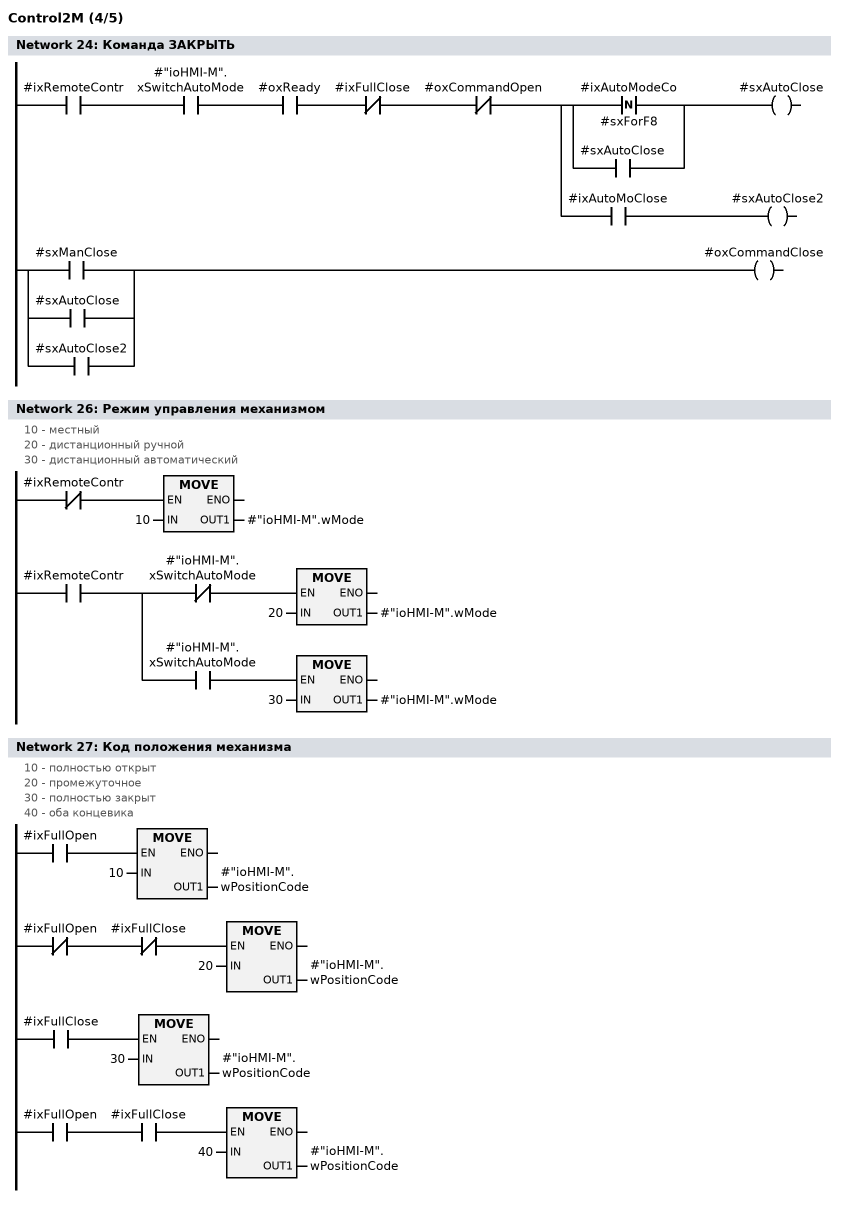
   RUNG wire#powerrail
      Contact( #ixRemoteContr )
      Contact( #"ioHMI-M".xSwitchAutoMode )
      Contact( #oxReady )
      I_Contact( #ixFullClose )
      I_Contact( #oxCommandOpen )
      wire#w1
      N_Contact(operand := #ixAutoModeCo, bit := #sxForF8)
      wire#w2
      Coil( #sxAutoClose )
   END_RUNG
   RUNG wire#w1
      Contact( #sxAutoClose )
   END_RUNG wire#w2
   RUNG wire#w1
      Contact( #ixAutoMoClose )
      Coil( #sxAutoClose2 )
   END_RUNG
   RUNG wire#powerrail
      Contact( #sxManClose )
      wire#w3
      Coil( #oxCommandClose )
   END_RUNG
   RUNG wire#powerrail
      Contact( #sxAutoClose )
   END_RUNG wire#w3
   RUNG wire#powerrail
      Contact( #sxAutoClose2 )
   END_RUNG wire#w3
   // the same network as SCL:
   #_w1 := #ixRemoteContr AND #"ioHMI-M".xSwitchAutoMode AND #oxReady AND NOT #ixFullClose AND NOT #oxCommandOpen;
   #_w2 := #_w1 AND NOT #ixAutoModeCo AND #sxForF8;   // falling edge of #ixAutoModeCo
   #sxForF8 := #ixAutoModeCo;
   #sxAutoClose := #_w2 OR (#_w1 AND #sxAutoClose);
   #sxAutoClose2 := #_w1 AND #ixAutoMoClose;
   #oxCommandClose := #sxManClose OR #sxAutoClose OR #sxAutoClose2;
END_REGION

REGION Network 26: Режим управления механизмом
   // 10 - местный
   // 20 - дистанционный ручной
   // 30 - дистанционный автоматический
   RUNG wire#powerrail
      I_Contact( #ixRemoteContr )
      Move(in := 10, out1 => #"ioHMI-M".wMode)
   END_RUNG
   RUNG wire#powerrail
      Contact( #ixRemoteContr )
      wire#w1
      I_Contact( #"ioHMI-M".xSwitchAutoMode )
      Move(in := 20, out1 => #"ioHMI-M".wMode)
   END_RUNG
   RUNG wire#w1
      Contact( #"ioHMI-M".xSwitchAutoMode )
      Move(in := 30, out1 => #"ioHMI-M".wMode)
   END_RUNG
   // the same network as SCL:
   IF NOT #ixRemoteContr THEN #"ioHMI-M".wMode := 10; END_IF;
   IF #ixRemoteContr AND NOT #"ioHMI-M".xSwitchAutoMode THEN #"ioHMI-M".wMode := 20; END_IF;
   IF #ixRemoteContr AND #"ioHMI-M".xSwitchAutoMode THEN #"ioHMI-M".wMode := 30; END_IF;
END_REGION

REGION Network 27: Код положения механизма
   // 10 - полностью открыт
   // 20 - промежуточное
   // 30 - полностью закрыт
   // 40 - оба концевика
   RUNG wire#powerrail
      Contact( #ixFullOpen )
      Move(in := 10, out1 => #"ioHMI-M".wPositionCode)
   END_RUNG
   RUNG wire#powerrail
      I_Contact( #ixFullOpen )
      I_Contact( #ixFullClose )
      Move(in := 20, out1 => #"ioHMI-M".wPositionCode)
   END_RUNG
   RUNG wire#powerrail
      Contact( #ixFullClose )
      Move(in := 30, out1 => #"ioHMI-M".wPositionCode)
   END_RUNG
   RUNG wire#powerrail
      Contact( #ixFullOpen )
      Contact( #ixFullClose )
      Move(in := 40, out1 => #"ioHMI-M".wPositionCode)
   END_RUNG
   // the same network as SCL:
   IF #ixFullOpen THEN #"ioHMI-M".wPositionCode := 10; END_IF;
   IF NOT #ixFullOpen AND NOT #ixFullClose THEN #"ioHMI-M".wPositionCode := 20; END_IF;
   IF #ixFullClose THEN #"ioHMI-M".wPositionCode := 30; END_IF;
   IF #ixFullOpen AND #ixFullClose THEN #"ioHMI-M".wPositionCode := 40; END_IF;
END_REGION

REGION Network 28: Код управления механизмом
   // 10 - нет команды на ход механизма
   // 20 - команда открыть
   // 30 - команда закрыть
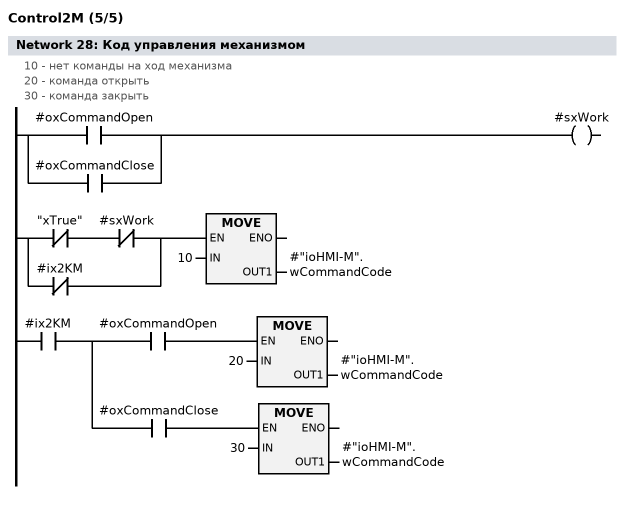
   RUNG wire#powerrail
      Contact( #oxCommandOpen )
      wire#w1
      Coil( #sxWork )
   END_RUNG
   RUNG wire#powerrail
      Contact( #oxCommandClose )
   END_RUNG wire#w1
   RUNG wire#powerrail
      I_Contact( "xTrue" )
      I_Contact( #sxWork )
      wire#w2
      Move(in := 10, out1 => #"ioHMI-M".wCommandCode)
   END_RUNG
   RUNG wire#powerrail
      I_Contact( #ix2KM )
   END_RUNG wire#w2
   RUNG wire#powerrail
      Contact( #ix2KM )
      wire#w3
      Contact( #oxCommandOpen )
      Move(in := 20, out1 => #"ioHMI-M".wCommandCode)
   END_RUNG
   RUNG wire#w3
      Contact( #oxCommandClose )
      Move(in := 30, out1 => #"ioHMI-M".wCommandCode)
   END_RUNG
   // the same network as SCL:
   #sxWork := #oxCommandOpen OR #oxCommandClose;
   IF (NOT "xTrue" AND NOT #sxWork) OR NOT #ix2KM THEN #"ioHMI-M".wCommandCode := 10; END_IF;
   IF #ix2KM AND #oxCommandOpen THEN #"ioHMI-M".wCommandCode := 20; END_IF;
   IF #ix2KM AND #oxCommandClose THEN #"ioHMI-M".wCommandCode := 30; END_IF;
END_REGION
END_FUNCTION_BLOCK

FUNCTION_BLOCK "ControlGate"   // FB503, LAD
{ S7_Optimized_Access := 'TRUE' }
VERSION : 0.1
   VAR_INPUT
      ixGateReady : Bool;   // Готовность шлюзового затвора
      ixRemoteContr : Bool;   // Ключ в положении Дистанц. рехим
      ixXKM : Bool;   // Пускатель включен
      ixExtStop : Bool;   // Внешняя блокировка
      ixAutoModeCommand : Bool;   // Авт.режим, 1=открыть, 0=закрыть
   END_VAR
   VAR_OUTPUT
      oxButSTART : Bool;   // Кнопка ПУСК ручного режима
      oxButSTOP : Bool;   // Кнопка СТОП ручного режима
      oxSwitchAutoMode : Bool;   // Переключатель (автомат.=1, ручной=0) на ЧМИ
      oxReady : Bool;   // Готовность механизма
      oxCommandOn : Bool;   // Команда Пуск
   END_VAR
   VAR_IN_OUT
      "ioHMI-M" : "uHMI-Machine";   // Структура данных связи с ЧМИ
   END_VAR
   VAR
      sxWarning : Bool;   // Есть предупреждения
      sxFault : Bool;   // Есть авария
      sxWork : Bool;   // Есть моя команда
      sxForF1 : Bool;   // Статический бит для обнаружения фронта сигнала
      sxForF6 : Bool;   // Статический бит для обнаружения фронта сигнала
      sxForF7 : Bool;   // Статический бит для обнаружения фронта сигнала
      IEC_TimerInstance2 : TON_TIME;   // Таймер
      IEC_TimerInstance1 : TON_TIME;   // Таймер
      sxManStart : Bool;   // Статический бит для команды ручного режима
      sxAutoStart : Bool;   // Статический бит для команды автоматического режима
   END_VAR
   VAR_TEMP
      tx1 : Bool;   // Временный бит
      tx2 : Bool;
   END_VAR
   VAR_TEMP   // added for the SCL form of the ladder/FBD networks
      _w1 : Bool;
      _w2 : Bool;
   END_VAR
BEGIN

REGION Network 4: Подготовка данных от HMI:
END_REGION

REGION Network 5 (SCL): -виртуальные кнопки
   #oxButSTART  :=  #"ioHMI-M".xButManOpen;
   #oxButSTOP :=  #"ioHMI-M".xButManClose;

   #oxSwitchAutoMode := #"ioHMI-M".xSwitchAutoMode;
END_REGION

REGION Network 7: ПРЕДУПРЕЖДЕНИЯ 3М-8М (для журнала предупреждений на ЧМИ)
   // //wWarnings.%X0 - полностью закрыт
   // //wWarnings.%X1 - полностью открыт
   // wWarnings.%X2 - нет готовности от механизма (было в дистанционном режиме, с 27.12.2020 - во всех режимах)
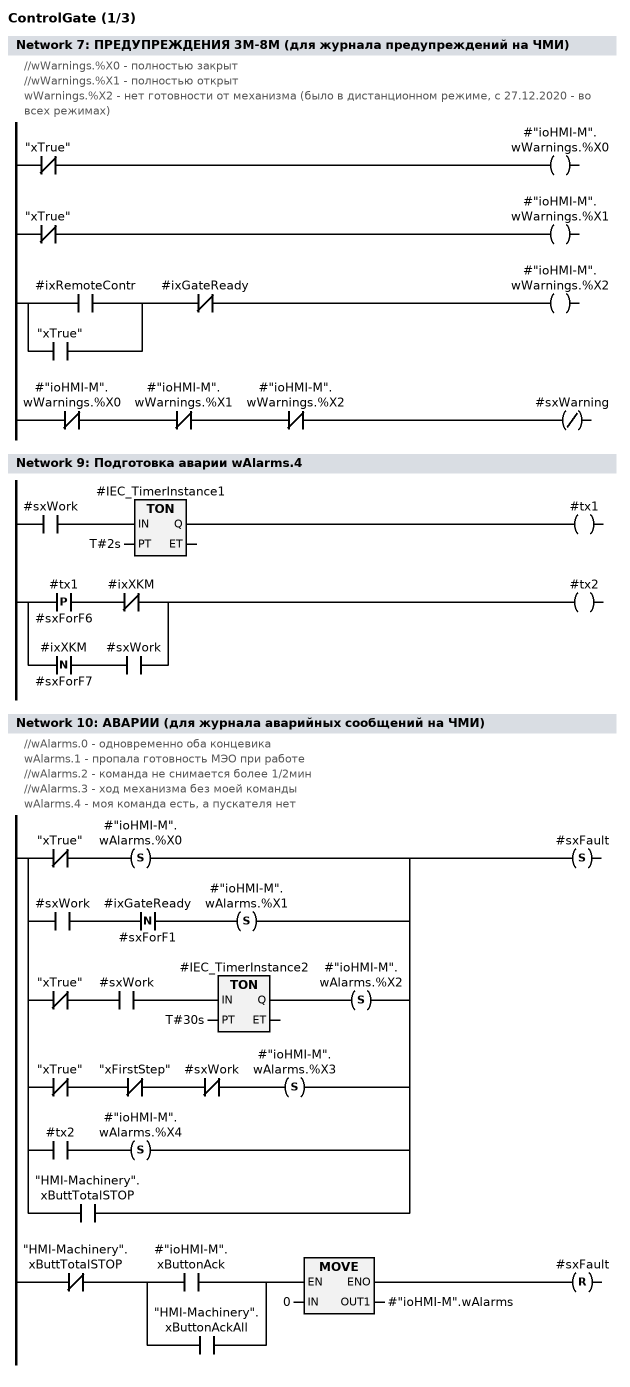
   RUNG wire#powerrail
      I_Contact( "xTrue" )
      Coil( #"ioHMI-M".wWarnings.%X0 )
   END_RUNG
   RUNG wire#powerrail
      I_Contact( "xTrue" )
      Coil( #"ioHMI-M".wWarnings.%X1 )
   END_RUNG
   RUNG wire#powerrail
      Contact( #ixRemoteContr )
      wire#w1
      I_Contact( #ixGateReady )
      Coil( #"ioHMI-M".wWarnings.%X2 )
   END_RUNG
   RUNG wire#powerrail
      Contact( "xTrue" )
   END_RUNG wire#w1
   RUNG wire#powerrail
      I_Contact( #"ioHMI-M".wWarnings.%X0 )
      I_Contact( #"ioHMI-M".wWarnings.%X1 )
      I_Contact( #"ioHMI-M".wWarnings.%X2 )
      I_Coil( #sxWarning )
   END_RUNG
   // the same network as SCL:
   #"ioHMI-M".wWarnings.%X0 := NOT "xTrue";
   #"ioHMI-M".wWarnings.%X1 := NOT "xTrue";
   #"ioHMI-M".wWarnings.%X2 := (#ixRemoteContr OR "xTrue") AND NOT #ixGateReady;
   #sxWarning := NOT (NOT #"ioHMI-M".wWarnings.%X0 AND NOT #"ioHMI-M".wWarnings.%X1 AND NOT #"ioHMI-M".wWarnings.%X2);
END_REGION

REGION Network 9: Подготовка аварии wAlarms.4
   #IEC_TimerInstance1(IN := #sxWork, PT := T#2s);   // TON
   #tx1 := #IEC_TimerInstance1.Q;
   #_w1 := #tx1 AND NOT #sxForF6;   // rising edge of #tx1
   #sxForF6 := #tx1;
   #_w2 := NOT #ixXKM AND #sxForF7;   // falling edge of #ixXKM
   #sxForF7 := #ixXKM;
   #tx2 := (#_w1 AND NOT #ixXKM) OR (#_w2 AND #sxWork);
END_REGION

REGION Network 10: АВАРИИ (для журнала аварийных сообщений на ЧМИ)
   // //wAlarms.0 - одновременно оба концевика
   // wAlarms.1 - пропала готовность МЭО при работе
   // //wAlarms.2 - команда не снимается более 1/2мин
   // //wAlarms.3 - ход механизма без моей команды 
   // wAlarms.4 - моя команда есть, а пускателя нет
   IF NOT "xTrue" THEN #"ioHMI-M".wAlarms.%X0 := TRUE; END_IF;
   #_w1 := #sxWork AND NOT #ixGateReady AND #sxForF1;   // falling edge of #ixGateReady
   #sxForF1 := #ixGateReady;
   IF #_w1 THEN #"ioHMI-M".wAlarms.%X1 := TRUE; END_IF;
   #IEC_TimerInstance2(IN := NOT "xTrue" AND #sxWork, PT := T#30s);   // TON
   IF #IEC_TimerInstance2.Q THEN #"ioHMI-M".wAlarms.%X2 := TRUE; END_IF;
   #_w2 := NOT "xTrue" AND NOT "xFirstStep" AND NOT #sxWork;
   IF #_w2 THEN #"ioHMI-M".wAlarms.%X3 := TRUE; END_IF;
   IF #tx2 THEN #"ioHMI-M".wAlarms.%X4 := TRUE; END_IF;
   IF NOT "xTrue" OR #_w1 OR #IEC_TimerInstance2.Q OR #_w2 OR #tx2 OR "HMI-Machinery".xButtTotalSTOP THEN
       #sxFault := TRUE;
   END_IF;
   IF NOT "HMI-Machinery".xButtTotalSTOP AND (#"ioHMI-M".xButtonAck OR "HMI-Machinery".xButtonAckAll) THEN
       #"ioHMI-M".wAlarms := 0;
       #sxFault := FALSE;
   END_IF;
END_REGION

REGION Network 12: Статус/состояние механизма:
END_REGION

REGION Network 13: -готов
   // 10 - готов
   // 20 - не готов
   // 30 - авария
   // 40 - внешняя блокировка
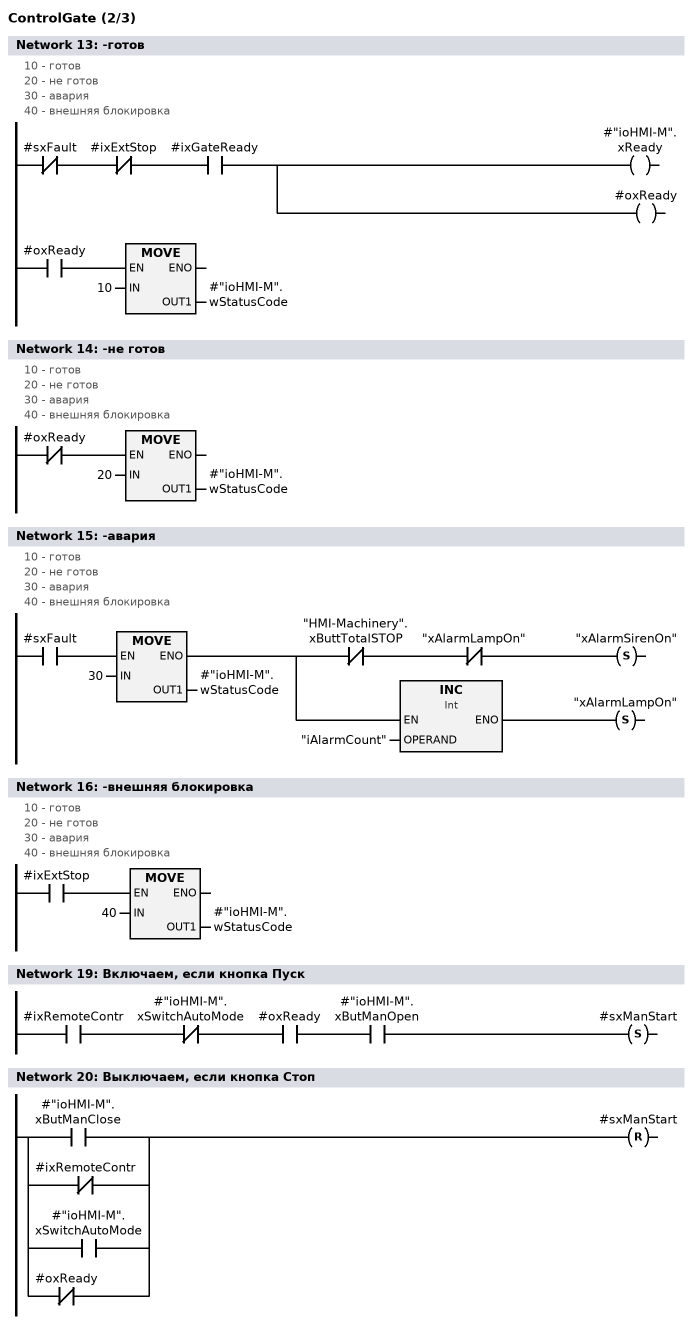
   RUNG wire#powerrail
      I_Contact( #sxFault )
      I_Contact( #ixExtStop )
      Contact( #ixGateReady )
      wire#w1
      Coil( #"ioHMI-M".xReady )
   END_RUNG
   RUNG wire#w1
      Coil( #oxReady )
   END_RUNG
   RUNG wire#powerrail
      Contact( #oxReady )
      Move(in := 10, out1 => #"ioHMI-M".wStatusCode)
   END_RUNG
   // the same network as SCL:
   #"ioHMI-M".xReady := NOT #sxFault AND NOT #ixExtStop AND #ixGateReady;
   #oxReady := #"ioHMI-M".xReady;
   IF #oxReady THEN #"ioHMI-M".wStatusCode := 10; END_IF;
END_REGION

REGION Network 14: -не готов
   // 10 - готов
   // 20 - не готов
   // 30 - авария
   // 40 - внешняя блокировка
   RUNG wire#powerrail
      I_Contact( #oxReady )
      Move(in := 20, out1 => #"ioHMI-M".wStatusCode)
   END_RUNG
   // the same network as SCL:
   IF NOT #oxReady THEN #"ioHMI-M".wStatusCode := 20; END_IF;
END_REGION

REGION Network 15: -авария
   // 10 - готов
   // 20 - не готов
   // 30 - авария
   // 40 - внешняя блокировка
   RUNG wire#powerrail
      Contact( #sxFault )
      Move(in := 30, out1 => #"ioHMI-M".wStatusCode)
      wire#w1
      I_Contact( "HMI-Machinery".xButtTotalSTOP )
      I_Contact( "xAlarmLampOn" )
      S_Coil( "xAlarmSirenOn" )
   END_RUNG
   RUNG wire#w1
      { S7_Templates := "DestType := Int" } Inc( "iAlarmCount" )
      S_Coil( "xAlarmLampOn" )
   END_RUNG
   // the same network as SCL:
   IF #sxFault THEN #"ioHMI-M".wStatusCode := 30; END_IF;
   IF #sxFault AND NOT "HMI-Machinery".xButtTotalSTOP AND NOT "xAlarmLampOn" THEN
       "xAlarmSirenOn" := TRUE;
   END_IF;
   IF #sxFault THEN
       "iAlarmCount" := "iAlarmCount" + 1;
       "xAlarmLampOn" := TRUE;
   END_IF;
END_REGION

REGION Network 16: -внешняя блокировка
   // 10 - готов
   // 20 - не готов
   // 30 - авария
   // 40 - внешняя блокировка
   RUNG wire#powerrail
      Contact( #ixExtStop )
      Move(in := 40, out1 => #"ioHMI-M".wStatusCode)
   END_RUNG
   // the same network as SCL:
   IF #ixExtStop THEN #"ioHMI-M".wStatusCode := 40; END_IF;
END_REGION

REGION Network 18: Дистанционный РУЧНОЙ:
END_REGION

REGION Network 19: Включаем, если кнопка Пуск
   RUNG wire#powerrail
      Contact( #ixRemoteContr )
      I_Contact( #"ioHMI-M".xSwitchAutoMode )
      Contact( #oxReady )
      Contact( #"ioHMI-M".xButManOpen )
      S_Coil( #sxManStart )
   END_RUNG
   // the same network as SCL:
   IF #ixRemoteContr AND NOT #"ioHMI-M".xSwitchAutoMode AND #oxReady AND #"ioHMI-M".xButManOpen THEN
       #sxManStart := TRUE;
   END_IF;
END_REGION

REGION Network 20: Выключаем, если кнопка Стоп
   RUNG wire#powerrail
      Contact( #"ioHMI-M".xButManClose )
      wire#w1
      R_Coil( #sxManStart )
   END_RUNG
   RUNG wire#powerrail
      I_Contact( #ixRemoteContr )
   END_RUNG wire#w1
   RUNG wire#powerrail
      Contact( #"ioHMI-M".xSwitchAutoMode )
   END_RUNG wire#w1
   RUNG wire#powerrail
      I_Contact( #oxReady )
   END_RUNG wire#w1
   // the same network as SCL:
   IF #"ioHMI-M".xButManClose OR NOT #ixRemoteContr OR #"ioHMI-M".xSwitchAutoMode OR NOT #oxReady THEN
       #sxManStart := FALSE;
   END_IF;
END_REGION

REGION Network 22: Дистанционный АВТОМАТИЧЕСКИЙ:
END_REGION

REGION Network 23: Команда ПУСК / СТОП
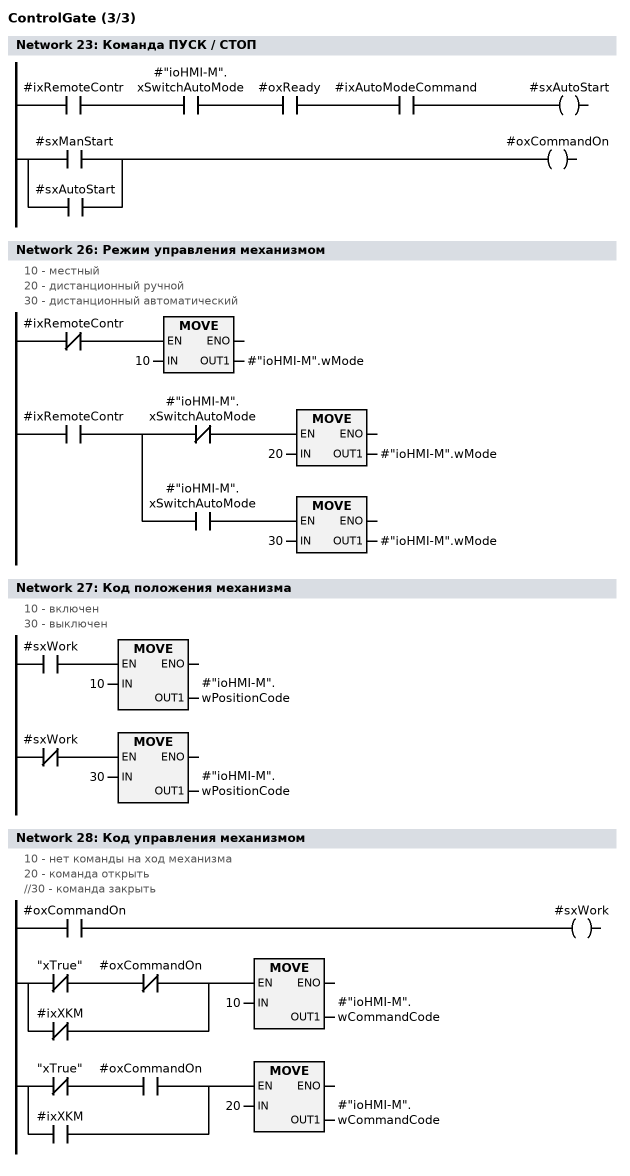
   RUNG wire#powerrail
      Contact( #ixRemoteContr )
      Contact( #"ioHMI-M".xSwitchAutoMode )
      Contact( #oxReady )
      Contact( #ixAutoModeCommand )
      Coil( #sxAutoStart )
   END_RUNG
   RUNG wire#powerrail
      Contact( #sxManStart )
      wire#w1
      Coil( #oxCommandOn )
   END_RUNG
   RUNG wire#powerrail
      Contact( #sxAutoStart )
   END_RUNG wire#w1
   // the same network as SCL:
   #sxAutoStart := #ixRemoteContr AND #"ioHMI-M".xSwitchAutoMode AND #oxReady AND #ixAutoModeCommand;
   #oxCommandOn := #sxManStart OR #sxAutoStart;
END_REGION

REGION Network 26: Режим управления механизмом
   // 10 - местный
   // 20 - дистанционный ручной
   // 30 - дистанционный автоматический
   RUNG wire#powerrail
      I_Contact( #ixRemoteContr )
      Move(in := 10, out1 => #"ioHMI-M".wMode)
   END_RUNG
   RUNG wire#powerrail
      Contact( #ixRemoteContr )
      wire#w1
      I_Contact( #"ioHMI-M".xSwitchAutoMode )
      Move(in := 20, out1 => #"ioHMI-M".wMode)
   END_RUNG
   RUNG wire#w1
      Contact( #"ioHMI-M".xSwitchAutoMode )
      Move(in := 30, out1 => #"ioHMI-M".wMode)
   END_RUNG
   // the same network as SCL:
   IF NOT #ixRemoteContr THEN #"ioHMI-M".wMode := 10; END_IF;
   IF #ixRemoteContr AND NOT #"ioHMI-M".xSwitchAutoMode THEN #"ioHMI-M".wMode := 20; END_IF;
   IF #ixRemoteContr AND #"ioHMI-M".xSwitchAutoMode THEN #"ioHMI-M".wMode := 30; END_IF;
END_REGION

REGION Network 27: Код положения механизма
   // 10 - включен
   // 30 - выключен
   RUNG wire#powerrail
      Contact( #sxWork )
      Move(in := 10, out1 => #"ioHMI-M".wPositionCode)
   END_RUNG
   RUNG wire#powerrail
      I_Contact( #sxWork )
      Move(in := 30, out1 => #"ioHMI-M".wPositionCode)
   END_RUNG
   // the same network as SCL:
   IF #sxWork THEN #"ioHMI-M".wPositionCode := 10; END_IF;
   IF NOT #sxWork THEN #"ioHMI-M".wPositionCode := 30; END_IF;
END_REGION

REGION Network 28: Код управления механизмом
   // 10 - нет команды на ход механизма
   // 20 - команда открыть
   // //30 - команда закрыть
   RUNG wire#powerrail
      Contact( #oxCommandOn )
      Coil( #sxWork )
   END_RUNG
   RUNG wire#powerrail
      I_Contact( "xTrue" )
      I_Contact( #oxCommandOn )
      wire#w1
      Move(in := 10, out1 => #"ioHMI-M".wCommandCode)
   END_RUNG
   RUNG wire#powerrail
      I_Contact( #ixXKM )
   END_RUNG wire#w1
   RUNG wire#powerrail
      I_Contact( "xTrue" )
      Contact( #oxCommandOn )
      wire#w2
      Move(in := 20, out1 => #"ioHMI-M".wCommandCode)
   END_RUNG
   RUNG wire#powerrail
      Contact( #ixXKM )
   END_RUNG wire#w2
   // the same network as SCL:
   #sxWork := #oxCommandOn;
   IF (NOT "xTrue" AND NOT #oxCommandOn) OR NOT #ixXKM THEN #"ioHMI-M".wCommandCode := 10; END_IF;
   IF (NOT "xTrue" AND #oxCommandOn) OR #ixXKM THEN #"ioHMI-M".wCommandCode := 20; END_IF;
END_REGION
END_FUNCTION_BLOCK

FUNCTION_BLOCK "ControlDym"   // FB509, LAD
{ S7_Optimized_Access := 'TRUE' }
VERSION : 0.1
   VAR_INPUT
      irSpeed : Real;   // Скорость двигателя
      ixDriveReady : Bool;   // Готовность привода дымососа
      ix2M_Ready : Bool;   // Готовность Направляющего аппарата
      ixPowerOn : Bool;   // Высокое напряжение подано
      ixLocalContr : Bool;   // Ключ в положении Местный рехим
      ixRemoteContr : Bool;   // Ключ в положении Дистанц. рехим
      ixDtiveFault : Bool;   // Авария привода=1, нет аварии=0
      ixExtStopTE102 : Bool;   // Внешняя блокировка по т-ре
      ixExtStopРІТ203 : Bool;   // Внешняя блокировка по разрежению
      ixExtStopVE : Bool;   // Внешняя блокировка по вибрации
      ixExtStopTEB : Bool;   // Внешняя блокировка по т-ре подшинников
      ixExtStopTEW : Bool;   // Внешняя блокировка по т-ре обмоток дв-ля
      ixLocalContrFbk : Bool;   // Выход привода Местный рехим
      ixRemoteContrFbk : Bool;   // Выход привода Дистанц. рехим
      ixWork : Bool;   // Сигнал Работа
   END_VAR
   VAR_OUTPUT
      oxButSTART : Bool;   // Кнопка СТАРТ
      oxButSTOP : Bool;   // Кнопка СТОП
      orSpeedGoTo : Real;   // Скорость для дистанционного ручного режима
      oxButGoTo : Bool;   // Кнопка Перехода На Заданую Скорость
      oxSwitchAutoMode : Bool;   // Переключатель (автомат.=1, ручной=0) на ЧМИ
      oxReady : Bool;   // Готовность механизма
      oxCommandSTART : Bool;   // Команда на привод Пуск
      oxCommandSTOP : Bool;   // Команда на привод Стоп: 0-стоп
   END_VAR
   VAR_IN_OUT
      "ioHMI-M" : "uHMI-Dym";   // Структура данных связи с ЧМИ
   END_VAR
   VAR
      sxWarning : Bool;   // Есть предупреждения
      sxFault : Bool;   // Есть авария=1, нет аварии=0
      sxWork : Bool;   // Есть моя команда
      sxForF1 : Bool;   // Статический бит для обнаружения фронта сигнала
      sxForF2 : Bool;   // Статический бит для обнаружения фронта сигнала
      sxForF3 : Bool;   // Статический бит для обнаружения фронта сигнала
      sxForF4 : Bool;   // Статический бит для обнаружения фронта сигнала
      sxGoTo : Bool;   // Бит Перехода На Заданую Скорость. Не исп.
      sxReadyMaxStart : Bool := 1;   // Готовность по числу пусков в час. Не исп.
      siNumStart : Int;   // Число пусков за текущий час. Не исп.
      siRef : Int;   // Задание скорости приводу для ЦАП
      IEC_Timer_0_Instance : TOF_TIME;   // Таймер
      sx1perc : Bool;   // Определение мин.скорости для числа пусков
      sxForF1perc : Bool;   // Статический бит для обнаружения фронта сигнала
      sx2perc : Bool;   // Определение макс.скорости для числа пусков
      sxForF2perc : Bool;   // Статический бит для обнаружения фронта сигнала
   END_VAR
   VAR_TEMP
      trRef : Real;   // Временная переменная типа Real
      tiRef : Int;   // Не исп.
      txMode : Bool;   // Временный бит
   END_VAR
   VAR_TEMP   // added for the SCL form of the ladder/FBD networks
      _w1 : Bool;
      _w2 : Bool;
   END_VAR
BEGIN

REGION Network 1: Подготовка данных для HMI:
END_REGION

REGION Network 2: -скорость двигателя
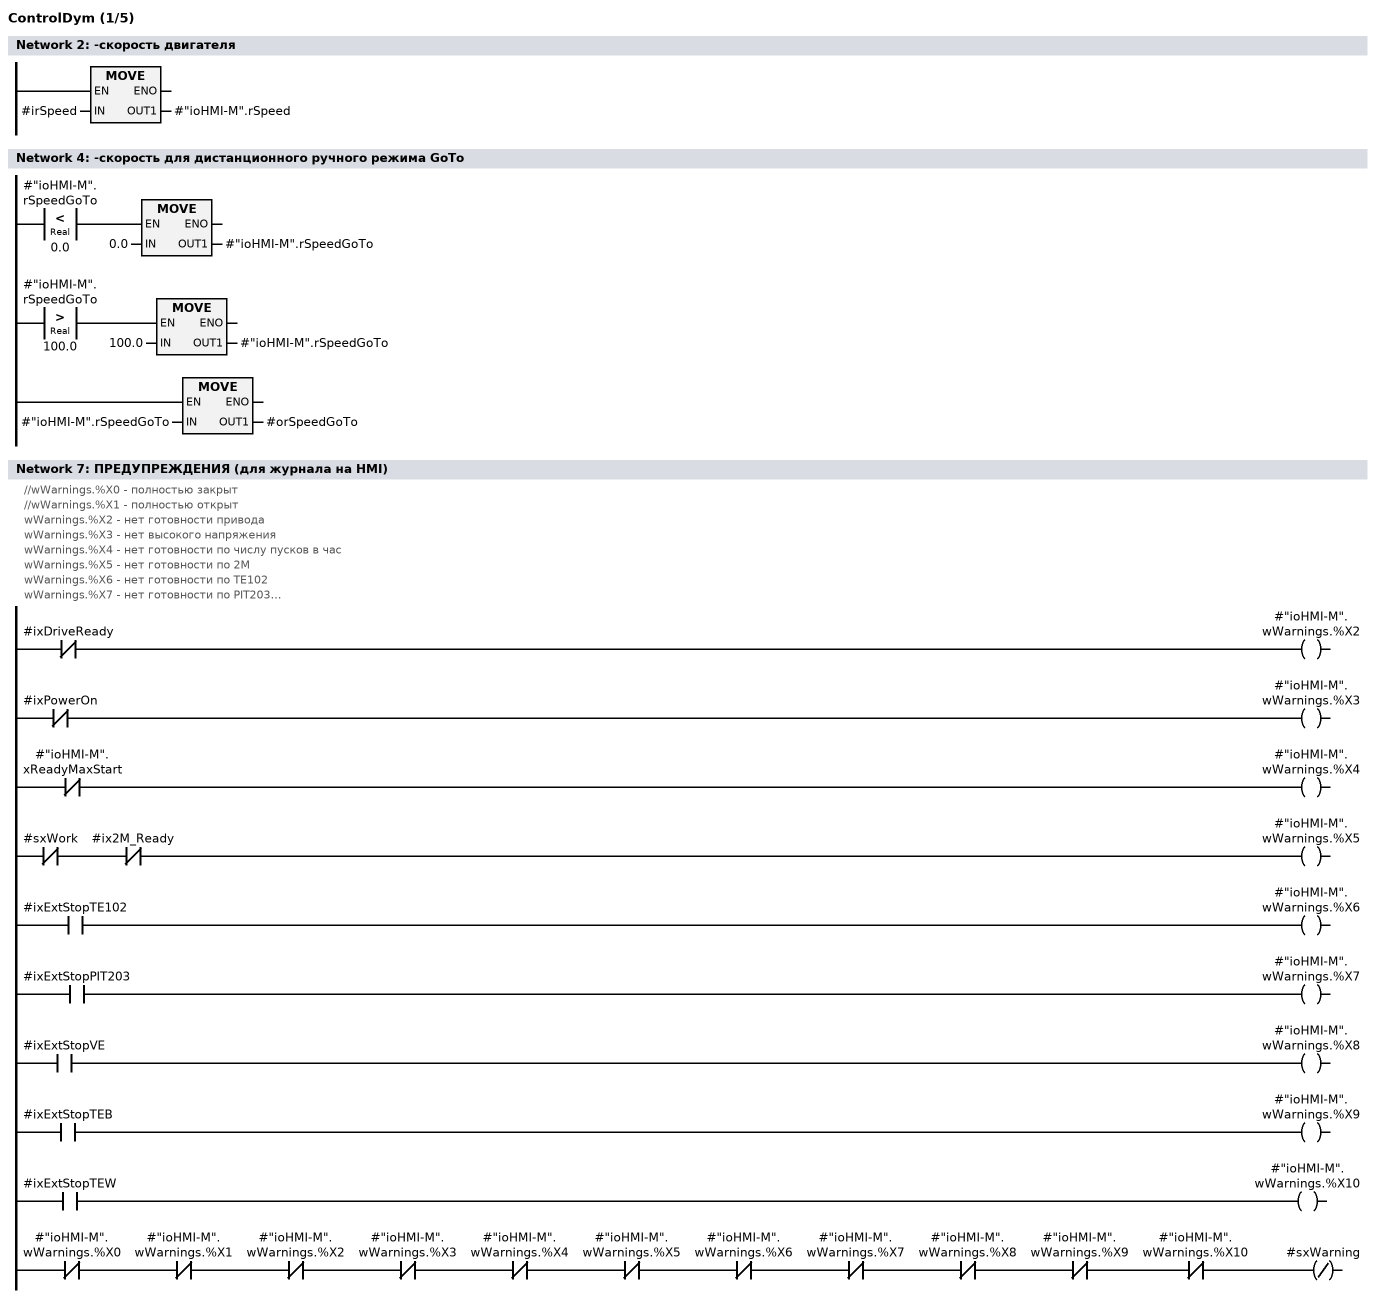
   RUNG wire#powerrail
      Move(in := #irSpeed, out1 => #"ioHMI-M".rSpeed)
   END_RUNG
   // the same network as SCL:
   #"ioHMI-M".rSpeed := #irSpeed;
END_REGION

REGION Network 3: Подготовка данных от HMI:
END_REGION

REGION Network 4: -скорость для дистанционного ручного режима GoTo
   RUNG wire#powerrail
      { S7_Templates := "SrcType := Real" } LT_Contact(in1 := #"ioHMI-M".rSpeedGoTo, in2 := 0.0)
      Move(in := 0.0, out1 => #"ioHMI-M".rSpeedGoTo)
   END_RUNG
   RUNG wire#powerrail
      { S7_Templates := "SrcType := Real" } GT_Contact(in1 := #"ioHMI-M".rSpeedGoTo, in2 := 100.0)
      Move(in := 100.0, out1 => #"ioHMI-M".rSpeedGoTo)
   END_RUNG
   RUNG wire#powerrail
      Move(in := #"ioHMI-M".rSpeedGoTo, out1 => #orSpeedGoTo)
   END_RUNG
   // the same network as SCL:
   IF #"ioHMI-M".rSpeedGoTo < 0.0 THEN #"ioHMI-M".rSpeedGoTo := 0.0; END_IF;
   IF #"ioHMI-M".rSpeedGoTo > 100.0 THEN #"ioHMI-M".rSpeedGoTo := 100.0; END_IF;
   #orSpeedGoTo := #"ioHMI-M".rSpeedGoTo;
END_REGION

REGION Network 5 (SCL): -виртуальные кнопки
   #oxButSTART :=  #"ioHMI-M".xButStart;
   #oxButSTOP  :=  #"ioHMI-M".xButStop;
   #oxButGoTo  :=  #"ioHMI-M".xButtonGoTo;
   #oxSwitchAutoMode := #"ioHMI-M".xSwitchAutoMode;
END_REGION

REGION Network 7: ПРЕДУПРЕЖДЕНИЯ (для журнала на НМІ)
   // //wWarnings.%X0 - полностью закрыт
   // //wWarnings.%X1 - полностью открыт
   // wWarnings.%X2 - нет готовности привода
   // wWarnings.%X3 - нет высокого напряжения 
   // wWarnings.%X4 - нет готовности по числу пусков в час
   // wWarnings.%X5 - нет готовности по 2М
   // wWarnings.%X6 - нет готовности по ТЕ102
   // wWarnings.%X7 - нет готовности по РІТ203, 
   // wWarnings.%X8 - нет готовности по вибрации
   // wWarnings.%X9 - нет готовности температуре подшипников
   // wWarnings.%Xa - нет готовности температуре обмоток
   RUNG wire#powerrail
      I_Contact( #ixDriveReady )
      Coil( #"ioHMI-M".wWarnings.%X2 )
   END_RUNG
   RUNG wire#powerrail
      I_Contact( #ixPowerOn )
      Coil( #"ioHMI-M".wWarnings.%X3 )
   END_RUNG
   RUNG wire#powerrail
      I_Contact( #"ioHMI-M".xReadyMaxStart )
      Coil( #"ioHMI-M".wWarnings.%X4 )
   END_RUNG
   RUNG wire#powerrail
      I_Contact( #sxWork )
      I_Contact( #ix2M_Ready )
      Coil( #"ioHMI-M".wWarnings.%X5 )
   END_RUNG
   RUNG wire#powerrail
      Contact( #ixExtStopTE102 )
      Coil( #"ioHMI-M".wWarnings.%X6 )
   END_RUNG
   RUNG wire#powerrail
      Contact( #ixExtStopРІТ203 )
      Coil( #"ioHMI-M".wWarnings.%X7 )
   END_RUNG
   RUNG wire#powerrail
      Contact( #ixExtStopVE )
      Coil( #"ioHMI-M".wWarnings.%X8 )
   END_RUNG
   RUNG wire#powerrail
      Contact( #ixExtStopTEB )
      Coil( #"ioHMI-M".wWarnings.%X9 )
   END_RUNG
   RUNG wire#powerrail
      Contact( #ixExtStopTEW )
      Coil( #"ioHMI-M".wWarnings.%X10 )
   END_RUNG
   RUNG wire#powerrail
      I_Contact( #"ioHMI-M".wWarnings.%X0 )
      I_Contact( #"ioHMI-M".wWarnings.%X1 )
      I_Contact( #"ioHMI-M".wWarnings.%X2 )
      I_Contact( #"ioHMI-M".wWarnings.%X3 )
      I_Contact( #"ioHMI-M".wWarnings.%X4 )
      I_Contact( #"ioHMI-M".wWarnings.%X5 )
      I_Contact( #"ioHMI-M".wWarnings.%X6 )
      I_Contact( #"ioHMI-M".wWarnings.%X7 )
      I_Contact( #"ioHMI-M".wWarnings.%X8 )
      I_Contact( #"ioHMI-M".wWarnings.%X9 )
      I_Contact( #"ioHMI-M".wWarnings.%X10 )
      I_Coil( #sxWarning )
   END_RUNG
   // the same network as SCL:
   #"ioHMI-M".wWarnings.%X2 := NOT #ixDriveReady;
   #"ioHMI-M".wWarnings.%X3 := NOT #ixPowerOn;
   #"ioHMI-M".wWarnings.%X4 := NOT #"ioHMI-M".xReadyMaxStart;
   #"ioHMI-M".wWarnings.%X5 := NOT #sxWork AND NOT #ix2M_Ready;
   #"ioHMI-M".wWarnings.%X6 := #ixExtStopTE102;
   #"ioHMI-M".wWarnings.%X7 := #ixExtStopРІТ203;
   #"ioHMI-M".wWarnings.%X8 := #ixExtStopVE;
   #"ioHMI-M".wWarnings.%X9 := #ixExtStopTEB;
   #"ioHMI-M".wWarnings.%X10 := #ixExtStopTEW;
   #sxWarning := NOT (NOT #"ioHMI-M".wWarnings.%X0 AND NOT #"ioHMI-M".wWarnings.%X1 AND NOT #"ioHMI-M".wWarnings.%X2 AND NOT #"ioHMI-M".wWarnings.%X3 AND NOT #"ioHMI-M".wWarnings.%X4 AND NOT #"ioHMI-M".wWarnings.%X5 AND NOT #"ioHMI-M".wWarnings.%X6 AND NOT #"ioHMI-M".wWarnings.%X7 AND NOT #"ioHMI-M".wWarnings.%X8 AND NOT #"ioHMI-M".wWarnings.%X9 AND NOT #"ioHMI-M".wWarnings.%X10);
END_REGION

REGION Network 10: АВАРИИ (для журнала аварийных сообщений на НМІ)
   // wAlarms.%X1 - пропала готовность дымососа при работе
   // wAlarms.%X6 - привод в ошибке
   // wAlarms.%X7 - внешний стоп по аварии блокирующих датчиков
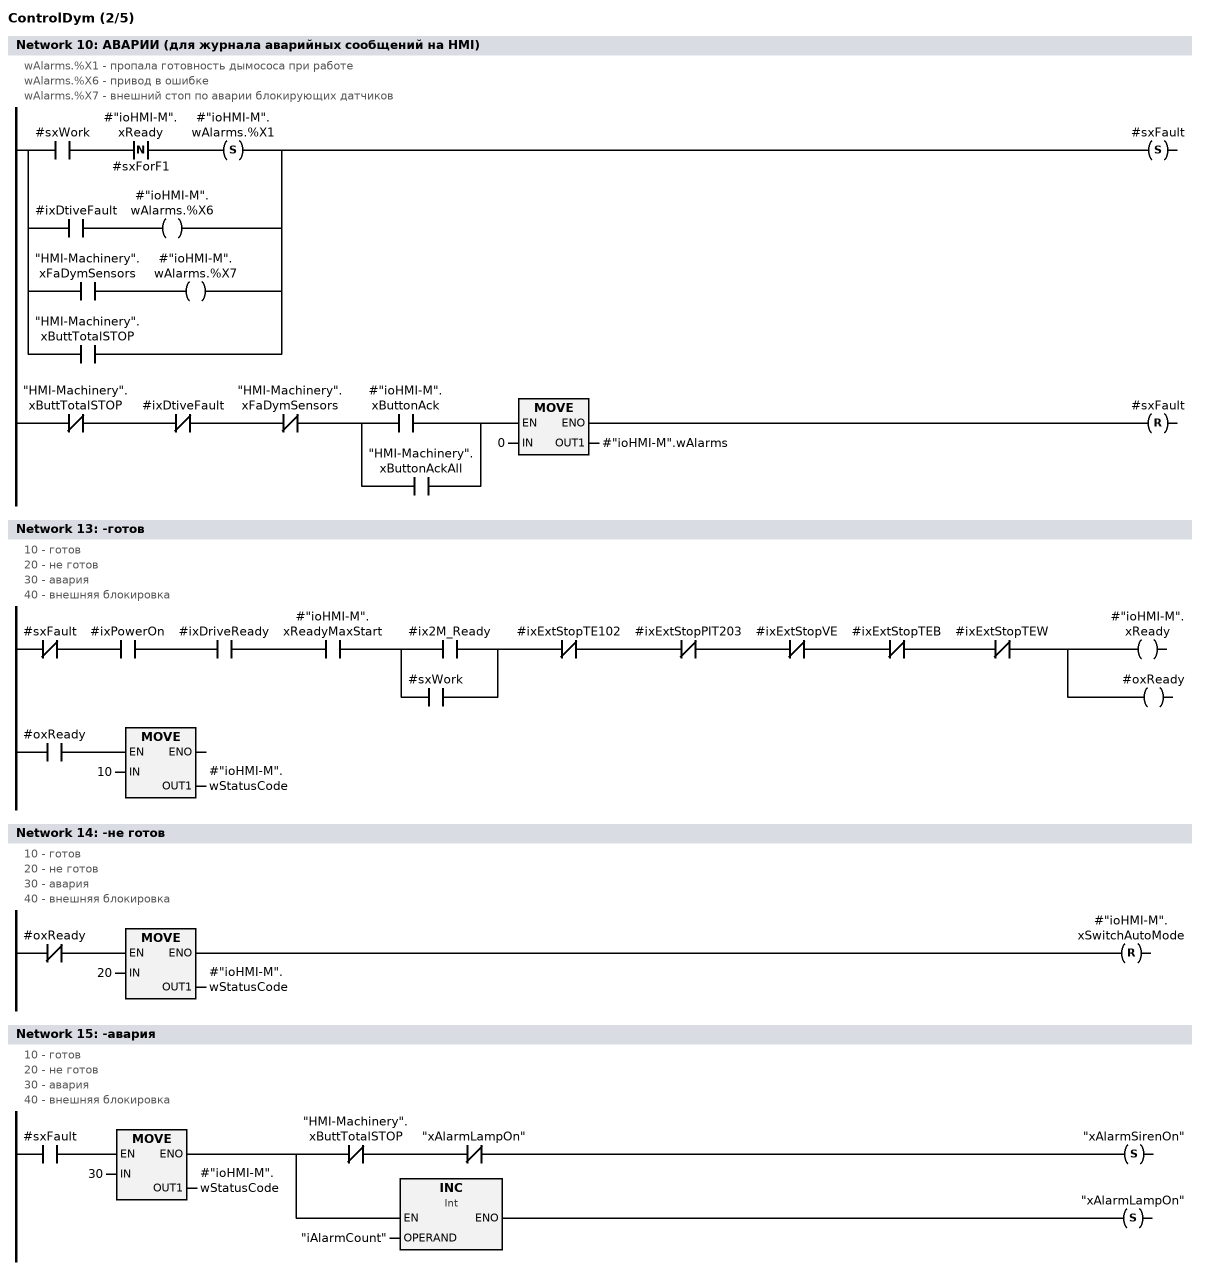
   RUNG wire#powerrail
      Contact( #sxWork )
      N_Contact(operand := #"ioHMI-M".xReady, bit := #sxForF1)
      S_Coil( #"ioHMI-M".wAlarms.%X1 )
      wire#w1
      S_Coil( #sxFault )
   END_RUNG
   RUNG wire#powerrail
      Contact( #ixDtiveFault )
      Coil( #"ioHMI-M".wAlarms.%X6 )
   END_RUNG wire#w1
   RUNG wire#powerrail
      Contact( "HMI-Machinery".xFaDymSensors )
      Coil( #"ioHMI-M".wAlarms.%X7 )
   END_RUNG wire#w1
   RUNG wire#powerrail
      Contact( "HMI-Machinery".xButtTotalSTOP )
   END_RUNG wire#w1
   RUNG wire#powerrail
      I_Contact( "HMI-Machinery".xButtTotalSTOP )
      I_Contact( #ixDtiveFault )
      I_Contact( "HMI-Machinery".xFaDymSensors )
      wire#w2
      Contact( #"ioHMI-M".xButtonAck )
      wire#w3
      Move(in := 0, out1 => #"ioHMI-M".wAlarms)
      R_Coil( #sxFault )
   END_RUNG
   RUNG wire#w2
      Contact( "HMI-Machinery".xButtonAckAll )
   END_RUNG wire#w3
   // the same network as SCL:
   #_w1 := #sxWork AND NOT #"ioHMI-M".xReady AND #sxForF1;   // falling edge of #"ioHMI-M".xReady
   #sxForF1 := #"ioHMI-M".xReady;
   IF #_w1 THEN #"ioHMI-M".wAlarms.%X1 := TRUE; END_IF;
   #"ioHMI-M".wAlarms.%X6 := #ixDtiveFault;
   #"ioHMI-M".wAlarms.%X7 := "HMI-Machinery".xFaDymSensors;
   IF #_w1 OR #ixDtiveFault OR "HMI-Machinery".xFaDymSensors OR "HMI-Machinery".xButtTotalSTOP THEN
       #sxFault := TRUE;
   END_IF;
   IF NOT "HMI-Machinery".xButtTotalSTOP AND NOT #ixDtiveFault AND NOT "HMI-Machinery".xFaDymSensors AND (#"ioHMI-M".xButtonAck OR "HMI-Machinery".xButtonAckAll) THEN
       #"ioHMI-M".wAlarms := 0;
       #sxFault := FALSE;
   END_IF;
END_REGION

REGION Network 12: Статус/состояние механизма:
END_REGION

REGION Network 13: -готов
   // 10 - готов
   // 20 - не готов
   // 30 - авария
   // 40 - внешняя блокировка
   RUNG wire#powerrail
      I_Contact( #sxFault )
      Contact( #ixPowerOn )
      Contact( #ixDriveReady )
      Contact( #"ioHMI-M".xReadyMaxStart )
      wire#w1
      Contact( #ix2M_Ready )
      wire#w2
      I_Contact( #ixExtStopTE102 )
      I_Contact( #ixExtStopРІТ203 )
      I_Contact( #ixExtStopVE )
      I_Contact( #ixExtStopTEB )
      I_Contact( #ixExtStopTEW )
      wire#w3
      Coil( #"ioHMI-M".xReady )
   END_RUNG
   RUNG wire#w1
      Contact( #sxWork )
   END_RUNG wire#w2
   RUNG wire#w3
      Coil( #oxReady )
   END_RUNG
   RUNG wire#powerrail
      Contact( #oxReady )
      Move(in := 10, out1 => #"ioHMI-M".wStatusCode)
   END_RUNG
   // the same network as SCL:
   #"ioHMI-M".xReady := NOT #sxFault AND #ixPowerOn AND #ixDriveReady AND #"ioHMI-M".xReadyMaxStart AND (#ix2M_Ready OR #sxWork) AND NOT #ixExtStopTE102 AND NOT #ixExtStopРІТ203 AND NOT #ixExtStopVE AND NOT #ixExtStopTEB AND NOT #ixExtStopTEW;
   #oxReady := #"ioHMI-M".xReady;
   IF #oxReady THEN #"ioHMI-M".wStatusCode := 10; END_IF;
END_REGION

REGION Network 14: -не готов
   // 10 - готов
   // 20 - не готов
   // 30 - авария
   // 40 - внешняя блокировка
   RUNG wire#powerrail
      I_Contact( #oxReady )
      Move(in := 20, out1 => #"ioHMI-M".wStatusCode)
      R_Coil( #"ioHMI-M".xSwitchAutoMode )
   END_RUNG
   // the same network as SCL:
   IF NOT #oxReady THEN
       #"ioHMI-M".wStatusCode := 20;
       #"ioHMI-M".xSwitchAutoMode := FALSE;
   END_IF;
END_REGION

REGION Network 15: -авария
   // 10 - готов
   // 20 - не готов
   // 30 - авария
   // 40 - внешняя блокировка
   RUNG wire#powerrail
      Contact( #sxFault )
      Move(in := 30, out1 => #"ioHMI-M".wStatusCode)
      wire#w1
      I_Contact( "HMI-Machinery".xButtTotalSTOP )
      I_Contact( "xAlarmLampOn" )
      S_Coil( "xAlarmSirenOn" )
   END_RUNG
   RUNG wire#w1
      { S7_Templates := "DestType := Int" } Inc( "iAlarmCount" )
      S_Coil( "xAlarmLampOn" )
   END_RUNG
   // the same network as SCL:
   IF #sxFault THEN #"ioHMI-M".wStatusCode := 30; END_IF;
   IF #sxFault AND NOT "HMI-Machinery".xButtTotalSTOP AND NOT "xAlarmLampOn" THEN
       "xAlarmSirenOn" := TRUE;
   END_IF;
   IF #sxFault THEN
       "iAlarmCount" := "iAlarmCount" + 1;
       "xAlarmLampOn" := TRUE;
   END_IF;
END_REGION

REGION Network 16: -внешняя блокировка
   // 10 - готов
   // 20 - не готов
   // 30 - авария
   // 40 - внешняя блокировка, отключено 14.01.2021
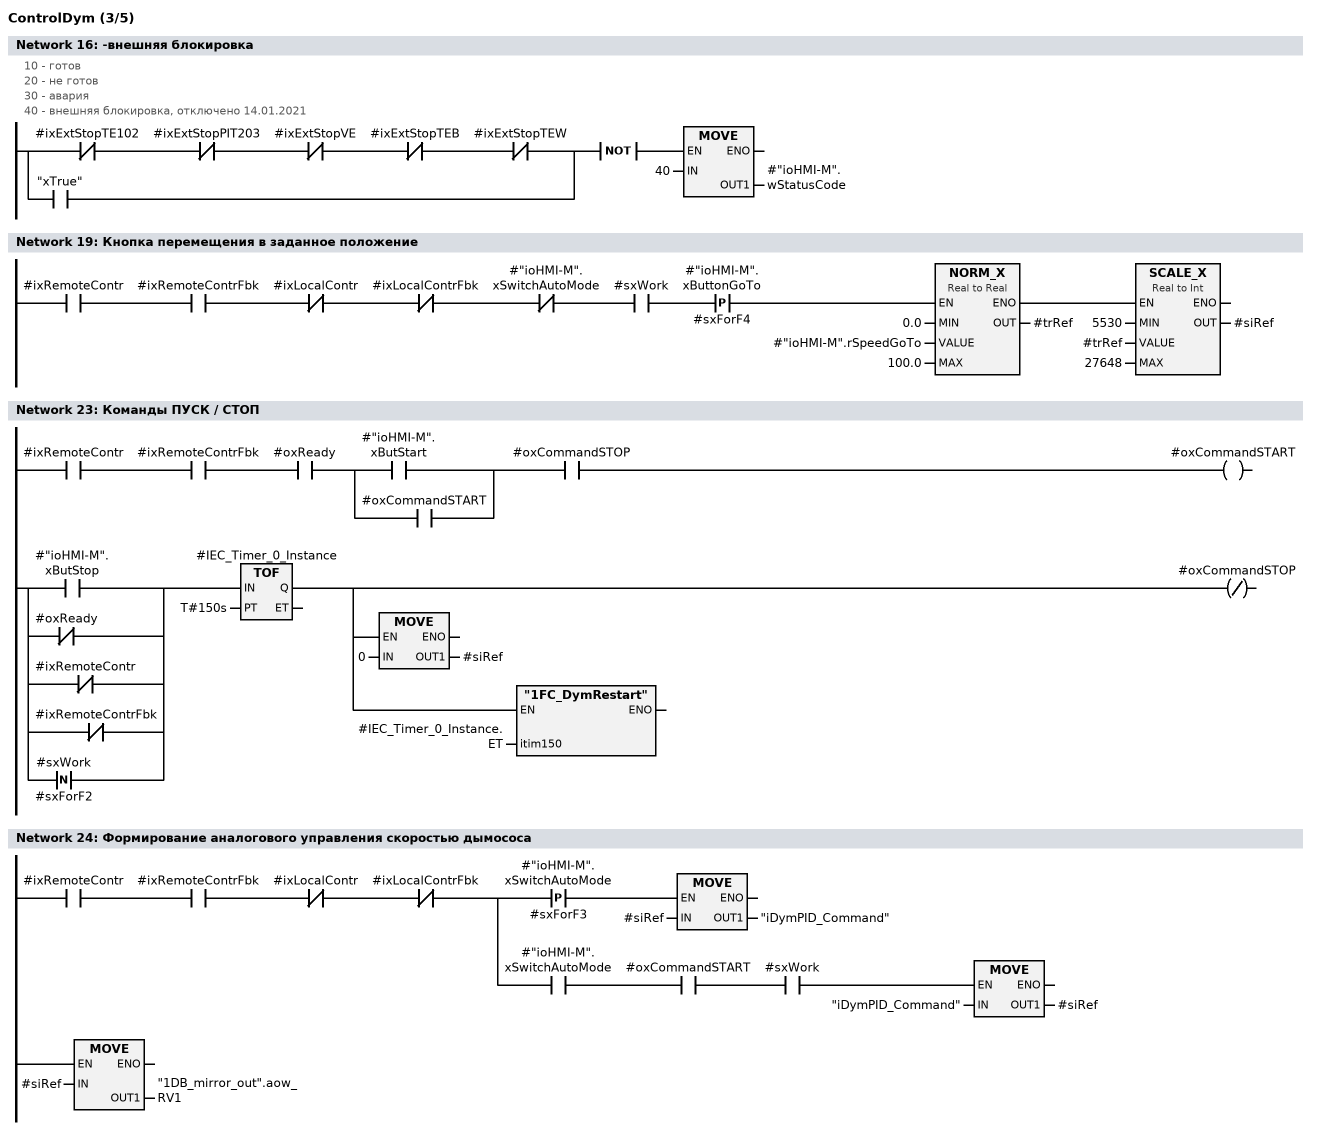
   RUNG wire#powerrail
      I_Contact( #ixExtStopTE102 )
      I_Contact( #ixExtStopРІТ203 )
      I_Contact( #ixExtStopVE )
      I_Contact( #ixExtStopTEB )
      I_Contact( #ixExtStopTEW )
      wire#w1
      Not()
      Move(in := 40, out1 => #"ioHMI-M".wStatusCode)
   END_RUNG
   RUNG wire#powerrail
      Contact( "xTrue" )
   END_RUNG wire#w1
   // the same network as SCL:
   IF NOT ((NOT #ixExtStopTE102 AND NOT #ixExtStopРІТ203 AND NOT #ixExtStopVE AND NOT #ixExtStopTEB AND NOT #ixExtStopTEW) OR "xTrue") THEN
       #"ioHMI-M".wStatusCode := 40;
   END_IF;
END_REGION

REGION Network 18: Дистанционный РУЧНОЙ:
END_REGION

REGION Network 19: Кнопка перемещения в заданное положение
   RUNG wire#powerrail
      Contact( #ixRemoteContr )
      Contact( #ixRemoteContrFbk )
      I_Contact( #ixLocalContr )
      I_Contact( #ixLocalContrFbk )
      I_Contact( #"ioHMI-M".xSwitchAutoMode )
      Contact( #sxWork )
      P_Contact(operand := #"ioHMI-M".xButtonGoTo, bit := #sxForF4)
      { S7_Templates := "[SrcType := Real, DestType := Real]" } Normalize(min := 0.0, value := #"ioHMI-M".rSpeedGoTo, max := 100.0, out => #trRef)
      { S7_Templates := "[SrcType := Real, DestType := Int]" } Scale(min := 5530, value := #trRef, max := 27648, out => #siRef)
   END_RUNG
   // the same network as SCL:
   #_w1 := #ixRemoteContr AND #ixRemoteContrFbk AND NOT #ixLocalContr AND NOT #ixLocalContrFbk AND NOT #"ioHMI-M".xSwitchAutoMode AND #sxWork AND #"ioHMI-M".xButtonGoTo AND NOT #sxForF4;   // rising edge of #"ioHMI-M".xButtonGoTo
   #sxForF4 := #"ioHMI-M".xButtonGoTo;
   IF #_w1 THEN
       #trRef := NORM_X(MIN := 0.0, VALUE := #"ioHMI-M".rSpeedGoTo, MAX := 100.0);
       #siRef := SCALE_X(MIN := 5530, VALUE := #trRef, MAX := 27648);
   END_IF;
END_REGION

REGION Network 22: Дистанционный (и ручной и автомат.):
END_REGION

REGION Network 23: Команды ПУСК / СТОП
   #oxCommandSTART := #ixRemoteContr AND #ixRemoteContrFbk AND #oxReady AND (#"ioHMI-M".xButStart OR #oxCommandSTART) AND #oxCommandSTOP;
   #_w1 := NOT #sxWork AND #sxForF2;   // falling edge of #sxWork
   #sxForF2 := #sxWork;
   #IEC_Timer_0_Instance(IN := #"ioHMI-M".xButStop OR NOT #oxReady OR NOT #ixRemoteContr OR NOT #ixRemoteContrFbk OR #_w1,   // TOF
                         PT := T#150s);
   #oxCommandSTOP := NOT #IEC_Timer_0_Instance.Q;
   IF #IEC_Timer_0_Instance.Q THEN
       #siRef := 0;
       "1FC_DymRestart"(itim150 := #IEC_Timer_0_Instance.ET);
   END_IF;
END_REGION

REGION Network 24: Формирование аналогового управления скоростью дымососа
   RUNG wire#powerrail
      Contact( #ixRemoteContr )
      Contact( #ixRemoteContrFbk )
      I_Contact( #ixLocalContr )
      I_Contact( #ixLocalContrFbk )
      wire#w1
      P_Contact(operand := #"ioHMI-M".xSwitchAutoMode, bit := #sxForF3)
      Move(in := #siRef, out1 => "iDymPID_Command")
   END_RUNG
   RUNG wire#w1
      Contact( #"ioHMI-M".xSwitchAutoMode )
      Contact( #oxCommandSTART )
      Contact( #sxWork )
      Move(in := "iDymPID_Command", out1 => #siRef)
   END_RUNG
   RUNG wire#powerrail
      Move(in := #siRef, out1 => "1DB_mirror_out".aow_RV1)
   END_RUNG
   // the same network as SCL:
   #_w1 := #ixRemoteContr AND #ixRemoteContrFbk AND NOT #ixLocalContr AND NOT #ixLocalContrFbk;
   #_w2 := #_w1 AND #"ioHMI-M".xSwitchAutoMode AND NOT #sxForF3;   // rising edge of #"ioHMI-M".xSwitchAutoMode
   #sxForF3 := #"ioHMI-M".xSwitchAutoMode;
   IF #_w2 THEN "iDymPID_Command" := #siRef; END_IF;
   IF #_w1 AND #"ioHMI-M".xSwitchAutoMode AND #oxCommandSTART AND #sxWork THEN
       #siRef := "iDymPID_Command";
   END_IF;
   "1DB_mirror_out".aow_RV1 := #siRef;
END_REGION

REGION Network 26: Режим управления механизмом
   // 10 - местный
   // 20 - дистанционный ручной
   // 30 - дистанционный автоматический
   // 40 - ошибка определения режима управления
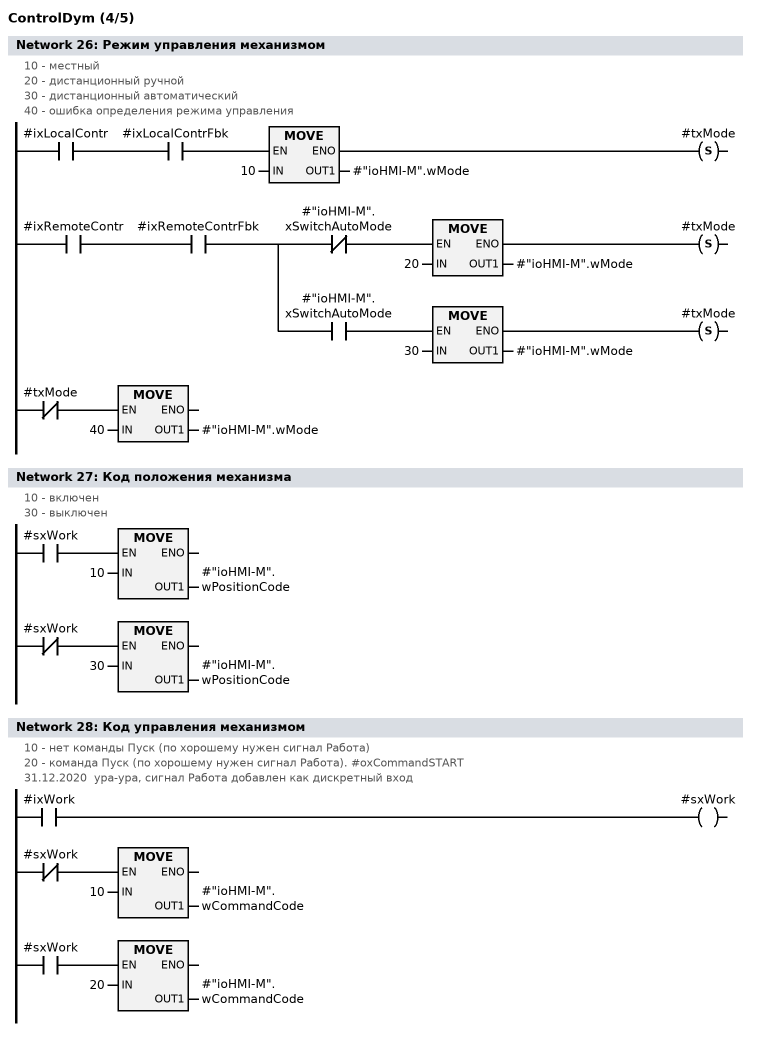
   RUNG wire#powerrail
      Contact( #ixLocalContr )
      Contact( #ixLocalContrFbk )
      Move(in := 10, out1 => #"ioHMI-M".wMode)
      S_Coil( #txMode )
   END_RUNG
   RUNG wire#powerrail
      Contact( #ixRemoteContr )
      Contact( #ixRemoteContrFbk )
      wire#w1
      I_Contact( #"ioHMI-M".xSwitchAutoMode )
      Move(in := 20, out1 => #"ioHMI-M".wMode)
      S_Coil( #txMode )
   END_RUNG
   RUNG wire#w1
      Contact( #"ioHMI-M".xSwitchAutoMode )
      Move(in := 30, out1 => #"ioHMI-M".wMode)
      S_Coil( #txMode )
   END_RUNG
   RUNG wire#powerrail
      I_Contact( #txMode )
      Move(in := 40, out1 => #"ioHMI-M".wMode)
   END_RUNG
   // the same network as SCL:
   IF #ixLocalContr AND #ixLocalContrFbk THEN
       #"ioHMI-M".wMode := 10;
       #txMode := TRUE;
   END_IF;
   #_w1 := #ixRemoteContr AND #ixRemoteContrFbk;
   IF #_w1 AND NOT #"ioHMI-M".xSwitchAutoMode THEN
       #"ioHMI-M".wMode := 20;
       #txMode := TRUE;
   END_IF;
   IF #_w1 AND #"ioHMI-M".xSwitchAutoMode THEN
       #"ioHMI-M".wMode := 30;
       #txMode := TRUE;
   END_IF;
   IF NOT #txMode THEN #"ioHMI-M".wMode := 40; END_IF;
END_REGION

REGION Network 27: Код положения механизма
   // 10 - включен
   // 30 - выключен
   RUNG wire#powerrail
      Contact( #sxWork )
      Move(in := 10, out1 => #"ioHMI-M".wPositionCode)
   END_RUNG
   RUNG wire#powerrail
      I_Contact( #sxWork )
      Move(in := 30, out1 => #"ioHMI-M".wPositionCode)
   END_RUNG
   // the same network as SCL:
   IF #sxWork THEN #"ioHMI-M".wPositionCode := 10; END_IF;
   IF NOT #sxWork THEN #"ioHMI-M".wPositionCode := 30; END_IF;
END_REGION

REGION Network 28: Код управления механизмом
   // 10 - нет команды Пуск (по хорошему нужен сигнал Работа)
   // 20 - команда Пуск (по хорошему нужен сигнал Работа). #oxCommandSTART
   // 31.12.2020  ура-ура, сигнал Работа добавлен как дискретный вход
   RUNG wire#powerrail
      Contact( #ixWork )
      Coil( #sxWork )
   END_RUNG
   RUNG wire#powerrail
      I_Contact( #sxWork )
      Move(in := 10, out1 => #"ioHMI-M".wCommandCode)
   END_RUNG
   RUNG wire#powerrail
      Contact( #sxWork )
      Move(in := 20, out1 => #"ioHMI-M".wCommandCode)
   END_RUNG
   // the same network as SCL:
   #sxWork := #ixWork;
   IF NOT #sxWork THEN #"ioHMI-M".wCommandCode := 10; END_IF;
   IF #sxWork THEN #"ioHMI-M".wCommandCode := 20; END_IF;
END_REGION

REGION Network 30: Число пусков инкрементируем, если скорость превысила 2%
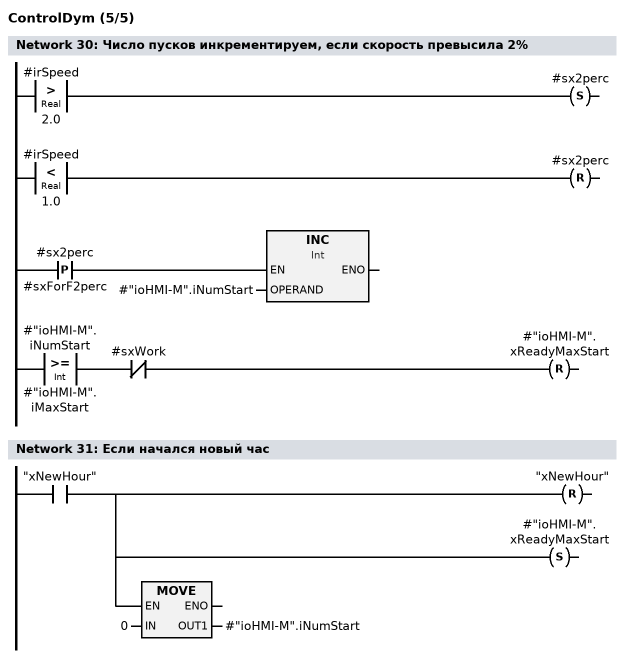
   RUNG wire#powerrail
      { S7_Templates := "SrcType := Real" } GT_Contact(in1 := #irSpeed, in2 := 2.0)
      S_Coil( #sx2perc )
   END_RUNG
   RUNG wire#powerrail
      { S7_Templates := "SrcType := Real" } LT_Contact(in1 := #irSpeed, in2 := 1.0)
      R_Coil( #sx2perc )
   END_RUNG
   RUNG wire#powerrail
      P_Contact(operand := #sx2perc, bit := #sxForF2perc)
      { S7_Templates := "DestType := Int" } Inc( #"ioHMI-M".iNumStart )
   END_RUNG
   RUNG wire#powerrail
      { S7_Templates := "SrcType := Int" } GE_Contact(in1 := #"ioHMI-M".iNumStart, in2 := #"ioHMI-M".iMaxStart)
      I_Contact( #sxWork )
      R_Coil( #"ioHMI-M".xReadyMaxStart )
   END_RUNG
   // the same network as SCL:
   IF #irSpeed > 2.0 THEN #sx2perc := TRUE; END_IF;
   IF #irSpeed < 1.0 THEN #sx2perc := FALSE; END_IF;
   #_w1 := #sx2perc AND NOT #sxForF2perc;   // rising edge of #sx2perc
   #sxForF2perc := #sx2perc;
   IF #_w1 THEN #"ioHMI-M".iNumStart := #"ioHMI-M".iNumStart + 1; END_IF;
   IF (#"ioHMI-M".iNumStart >= #"ioHMI-M".iMaxStart) AND NOT #sxWork THEN
       #"ioHMI-M".xReadyMaxStart := FALSE;
   END_IF;
END_REGION

REGION Network 31: Если начался новый час
   RUNG wire#powerrail
      Contact( "xNewHour" )
      wire#w1
      R_Coil( "xNewHour" )
   END_RUNG
   RUNG wire#w1
      S_Coil( #"ioHMI-M".xReadyMaxStart )
   END_RUNG
   RUNG wire#w1
      Move(in := 0, out1 => #"ioHMI-M".iNumStart)
   END_RUNG
   // the same network as SCL:
   #_w1 := "xNewHour";
   IF #_w1 THEN
       "xNewHour" := FALSE;
       #"ioHMI-M".xReadyMaxStart := TRUE;
       #"ioHMI-M".iNumStart := 0;
   END_IF;
END_REGION
END_FUNCTION_BLOCK

FUNCTION "GATEs" : Void   // FC503, LAD
{ S7_Optimized_Access := 'TRUE' }
VERSION : 0.1
// Управление шлюзовыми затворами
BEGIN

REGION Network 3: Затвор шлюзовый 3М
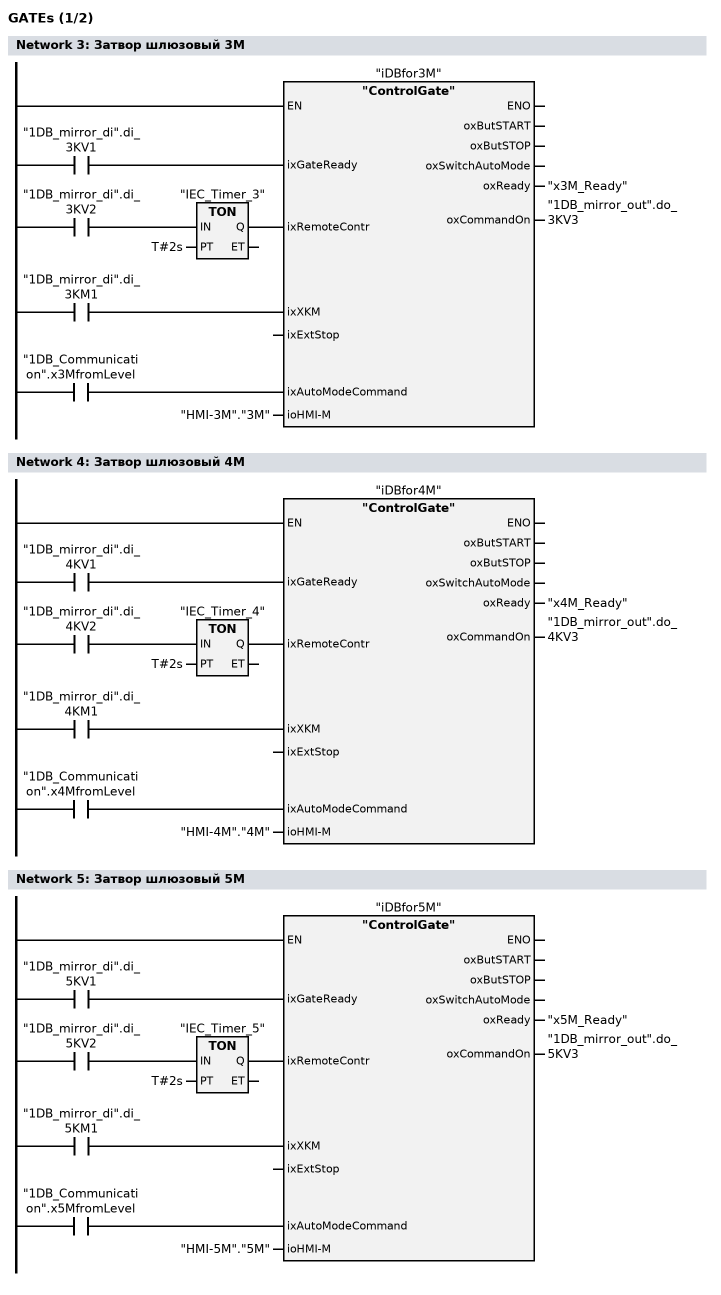
   "IEC_Timer_3".TON(IN := "1DB_mirror_di".di_3KV2, PT := T#2s);
   "iDBfor3M"(ixGateReady := "1DB_mirror_di".di_3KV1,   // "ControlGate"
              ixRemoteContr := "IEC_Timer_3".Q,
              ixXKM := "1DB_mirror_di".di_3KM1,
              ixAutoModeCommand := "1DB_Communication".x3MfromLevel,
              "ioHMI-M" := "HMI-3M"."3M",
              oxReady => "x3M_Ready",
              oxCommandOn => "1DB_mirror_out".do_3KV3);
END_REGION

REGION Network 4: Затвор шлюзовый 4М
   "IEC_Timer_4".TON(IN := "1DB_mirror_di".di_4KV2, PT := T#2s);
   "iDBfor4M"(ixGateReady := "1DB_mirror_di".di_4KV1,   // "ControlGate"
              ixRemoteContr := "IEC_Timer_4".Q,
              ixXKM := "1DB_mirror_di".di_4KM1,
              ixAutoModeCommand := "1DB_Communication".x4MfromLevel,
              "ioHMI-M" := "HMI-4M"."4M",
              oxReady => "x4M_Ready",
              oxCommandOn => "1DB_mirror_out".do_4KV3);
END_REGION

REGION Network 5: Затвор шлюзовый 5М
   "IEC_Timer_5".TON(IN := "1DB_mirror_di".di_5KV2, PT := T#2s);
   "iDBfor5M"(ixGateReady := "1DB_mirror_di".di_5KV1,   // "ControlGate"
              ixRemoteContr := "IEC_Timer_5".Q,
              ixXKM := "1DB_mirror_di".di_5KM1,
              ixAutoModeCommand := "1DB_Communication".x5MfromLevel,
              "ioHMI-M" := "HMI-5M"."5M",
              oxReady => "x5M_Ready",
              oxCommandOn => "1DB_mirror_out".do_5KV3);
END_REGION

REGION Network 6: Затвор шлюзовый 6М
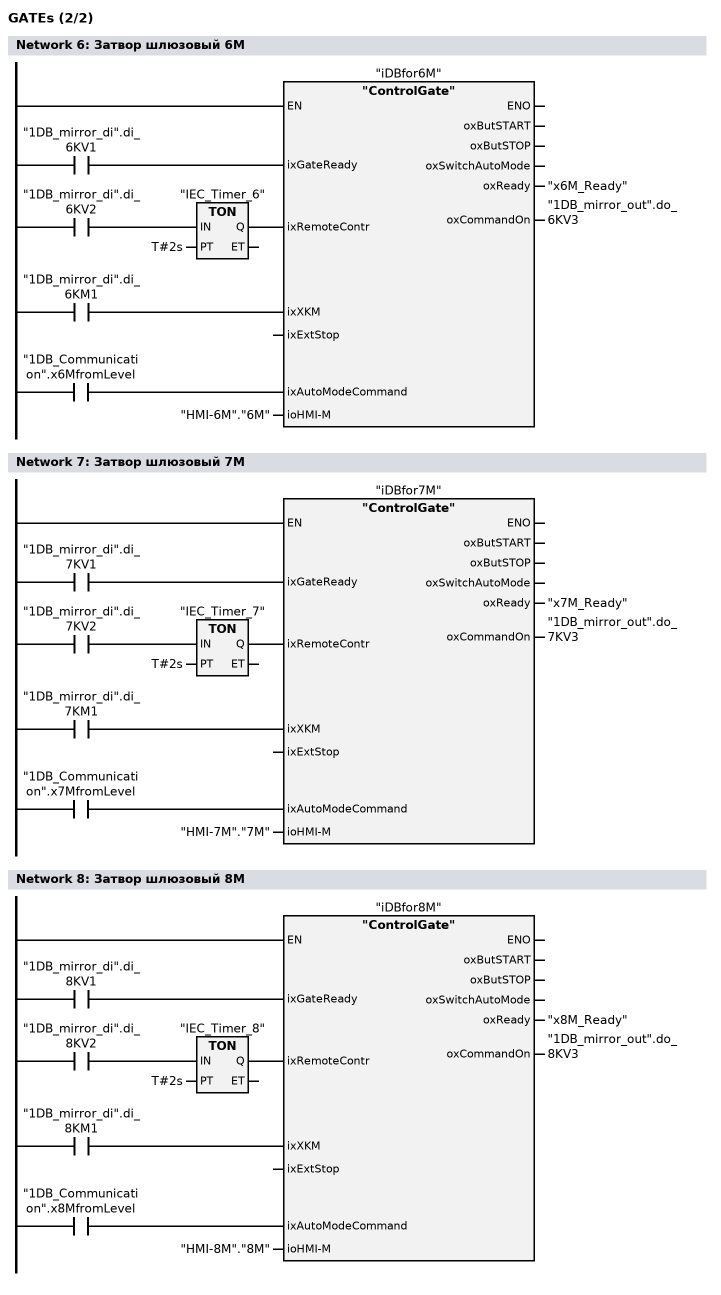
   "IEC_Timer_6".TON(IN := "1DB_mirror_di".di_6KV2, PT := T#2s);
   "iDBfor6M"(ixGateReady := "1DB_mirror_di".di_6KV1,   // "ControlGate"
              ixRemoteContr := "IEC_Timer_6".Q,
              ixXKM := "1DB_mirror_di".di_6KM1,
              ixAutoModeCommand := "1DB_Communication".x6MfromLevel,
              "ioHMI-M" := "HMI-6M"."6M",
              oxReady => "x6M_Ready",
              oxCommandOn => "1DB_mirror_out".do_6KV3);
END_REGION

REGION Network 7: Затвор шлюзовый 7М
   "IEC_Timer_7".TON(IN := "1DB_mirror_di".di_7KV2, PT := T#2s);
   "iDBfor7M"(ixGateReady := "1DB_mirror_di".di_7KV1,   // "ControlGate"
              ixRemoteContr := "IEC_Timer_7".Q,
              ixXKM := "1DB_mirror_di".di_7KM1,
              ixAutoModeCommand := "1DB_Communication".x7MfromLevel,
              "ioHMI-M" := "HMI-7M"."7M",
              oxReady => "x7M_Ready",
              oxCommandOn => "1DB_mirror_out".do_7KV3);
END_REGION

REGION Network 8: Затвор шлюзовый 8М
   "IEC_Timer_8".TON(IN := "1DB_mirror_di".di_8KV2, PT := T#2s);
   "iDBfor8M"(ixGateReady := "1DB_mirror_di".di_8KV1,   // "ControlGate"
              ixRemoteContr := "IEC_Timer_8".Q,
              ixXKM := "1DB_mirror_di".di_8KM1,
              ixAutoModeCommand := "1DB_Communication".x8MfromLevel,
              "ioHMI-M" := "HMI-8M"."8M",
              oxReady => "x8M_Ready",
              oxCommandOn => "1DB_mirror_out".do_8KV3);
END_REGION
END_FUNCTION

// folder: Mirrors

FUNCTION "1FC_mirroring_aiw" : Void   // FC101, LAD
{ S7_Optimized_Access := 'TRUE' }
VERSION : 0.1
BEGIN

REGION Network 2: Заполнение DB101 аналоговыми входами из модуля А1.02
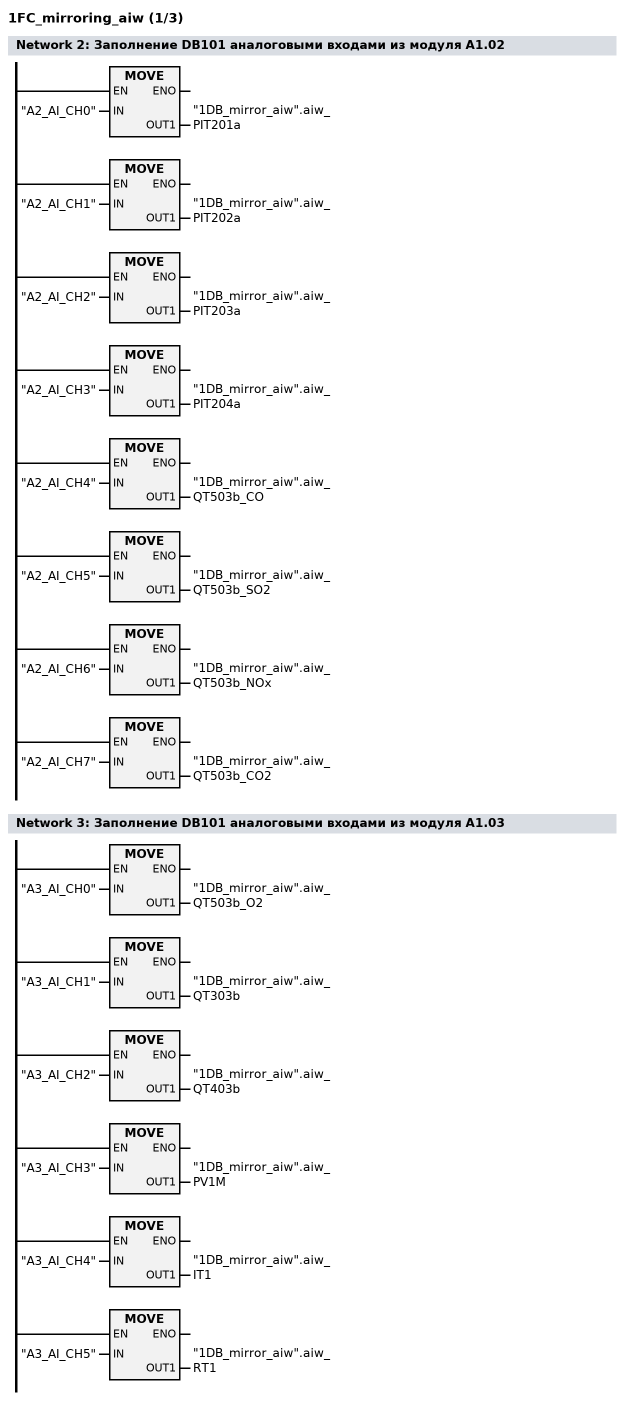
   RUNG wire#powerrail
      Move(in := "A2_AI_CH0", out1 => "1DB_mirror_aiw".aiw_PIT201a)
   END_RUNG
   RUNG wire#powerrail
      Move(in := "A2_AI_CH1", out1 => "1DB_mirror_aiw".aiw_PIT202a)
   END_RUNG
   RUNG wire#powerrail
      Move(in := "A2_AI_CH2", out1 => "1DB_mirror_aiw".aiw_PIT203a)
   END_RUNG
   RUNG wire#powerrail
      Move(in := "A2_AI_CH3", out1 => "1DB_mirror_aiw".aiw_PIT204a)
   END_RUNG
   RUNG wire#powerrail
      Move(in := "A2_AI_CH4", out1 => "1DB_mirror_aiw".aiw_QT503b_CO)
   END_RUNG
   RUNG wire#powerrail
      Move(in := "A2_AI_CH5", out1 => "1DB_mirror_aiw".aiw_QT503b_SO2)
   END_RUNG
   RUNG wire#powerrail
      Move(in := "A2_AI_CH6", out1 => "1DB_mirror_aiw".aiw_QT503b_NOx)
   END_RUNG
   RUNG wire#powerrail
      Move(in := "A2_AI_CH7", out1 => "1DB_mirror_aiw".aiw_QT503b_CO2)
   END_RUNG
   // the same network as SCL:
   "1DB_mirror_aiw".aiw_PIT201a := "A2_AI_CH0";
   "1DB_mirror_aiw".aiw_PIT202a := "A2_AI_CH1";
   "1DB_mirror_aiw".aiw_PIT203a := "A2_AI_CH2";
   "1DB_mirror_aiw".aiw_PIT204a := "A2_AI_CH3";
   "1DB_mirror_aiw".aiw_QT503b_CO := "A2_AI_CH4";
   "1DB_mirror_aiw".aiw_QT503b_SO2 := "A2_AI_CH5";
   "1DB_mirror_aiw".aiw_QT503b_NOx := "A2_AI_CH6";
   "1DB_mirror_aiw".aiw_QT503b_CO2 := "A2_AI_CH7";
END_REGION

REGION Network 3: Заполнение DB101 аналоговыми входами из модуля А1.03
   RUNG wire#powerrail
      Move(in := "A3_AI_CH0", out1 => "1DB_mirror_aiw".aiw_QT503b_O2)
   END_RUNG
   RUNG wire#powerrail
      Move(in := "A3_AI_CH1", out1 => "1DB_mirror_aiw".aiw_QT303b)
   END_RUNG
   RUNG wire#powerrail
      Move(in := "A3_AI_CH2", out1 => "1DB_mirror_aiw".aiw_QT403b)
   END_RUNG
   RUNG wire#powerrail
      Move(in := "A3_AI_CH3", out1 => "1DB_mirror_aiw".aiw_PV1M)
   END_RUNG
   RUNG wire#powerrail
      Move(in := "A3_AI_CH4", out1 => "1DB_mirror_aiw".aiw_IT1)
   END_RUNG
   RUNG wire#powerrail
      Move(in := "A3_AI_CH5", out1 => "1DB_mirror_aiw".aiw_RT1)
   END_RUNG
   // the same network as SCL:
   "1DB_mirror_aiw".aiw_QT503b_O2 := "A3_AI_CH0";
   "1DB_mirror_aiw".aiw_QT303b := "A3_AI_CH1";
   "1DB_mirror_aiw".aiw_QT403b := "A3_AI_CH2";
   "1DB_mirror_aiw".aiw_PV1M := "A3_AI_CH3";
   "1DB_mirror_aiw".aiw_IT1 := "A3_AI_CH4";
   "1DB_mirror_aiw".aiw_RT1 := "A3_AI_CH5";
END_REGION

REGION Network 4: Заполнение DB101 аналоговыми входами из модуля А1.04
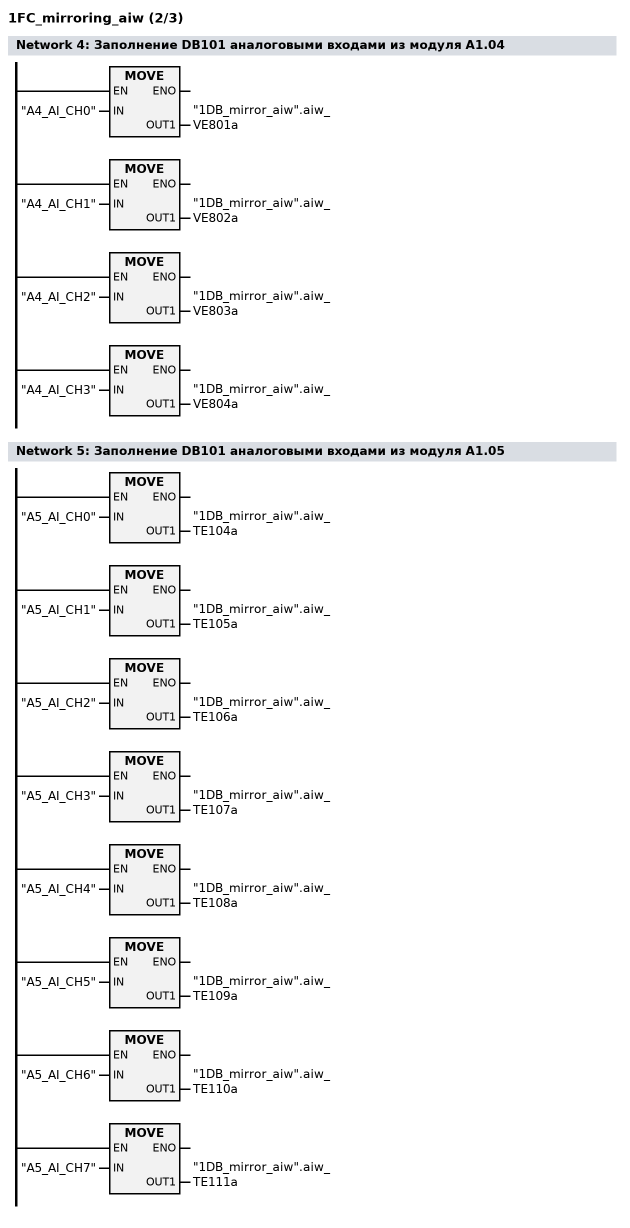
   RUNG wire#powerrail
      Move(in := "A4_AI_CH0", out1 => "1DB_mirror_aiw".aiw_VE801a)
   END_RUNG
   RUNG wire#powerrail
      Move(in := "A4_AI_CH1", out1 => "1DB_mirror_aiw".aiw_VE802a)
   END_RUNG
   RUNG wire#powerrail
      Move(in := "A4_AI_CH2", out1 => "1DB_mirror_aiw".aiw_VE803a)
   END_RUNG
   RUNG wire#powerrail
      Move(in := "A4_AI_CH3", out1 => "1DB_mirror_aiw".aiw_VE804a)
   END_RUNG
   // the same network as SCL:
   "1DB_mirror_aiw".aiw_VE801a := "A4_AI_CH0";
   "1DB_mirror_aiw".aiw_VE802a := "A4_AI_CH1";
   "1DB_mirror_aiw".aiw_VE803a := "A4_AI_CH2";
   "1DB_mirror_aiw".aiw_VE804a := "A4_AI_CH3";
END_REGION

REGION Network 5: Заполнение DB101 аналоговыми входами из модуля А1.05
   RUNG wire#powerrail
      Move(in := "A5_AI_CH0", out1 => "1DB_mirror_aiw".aiw_TE104a)
   END_RUNG
   RUNG wire#powerrail
      Move(in := "A5_AI_CH1", out1 => "1DB_mirror_aiw".aiw_TE105a)
   END_RUNG
   RUNG wire#powerrail
      Move(in := "A5_AI_CH2", out1 => "1DB_mirror_aiw".aiw_TE106a)
   END_RUNG
   RUNG wire#powerrail
      Move(in := "A5_AI_CH3", out1 => "1DB_mirror_aiw".aiw_TE107a)
   END_RUNG
   RUNG wire#powerrail
      Move(in := "A5_AI_CH4", out1 => "1DB_mirror_aiw".aiw_TE108a)
   END_RUNG
   RUNG wire#powerrail
      Move(in := "A5_AI_CH5", out1 => "1DB_mirror_aiw".aiw_TE109a)
   END_RUNG
   RUNG wire#powerrail
      Move(in := "A5_AI_CH6", out1 => "1DB_mirror_aiw".aiw_TE110a)
   END_RUNG
   RUNG wire#powerrail
      Move(in := "A5_AI_CH7", out1 => "1DB_mirror_aiw".aiw_TE111a)
   END_RUNG
   // the same network as SCL:
   "1DB_mirror_aiw".aiw_TE104a := "A5_AI_CH0";
   "1DB_mirror_aiw".aiw_TE105a := "A5_AI_CH1";
   "1DB_mirror_aiw".aiw_TE106a := "A5_AI_CH2";
   "1DB_mirror_aiw".aiw_TE107a := "A5_AI_CH3";
   "1DB_mirror_aiw".aiw_TE108a := "A5_AI_CH4";
   "1DB_mirror_aiw".aiw_TE109a := "A5_AI_CH5";
   "1DB_mirror_aiw".aiw_TE110a := "A5_AI_CH6";
   "1DB_mirror_aiw".aiw_TE111a := "A5_AI_CH7";
END_REGION

REGION Network 6: Заполнение DB101 аналоговыми входами из модуля А1.06
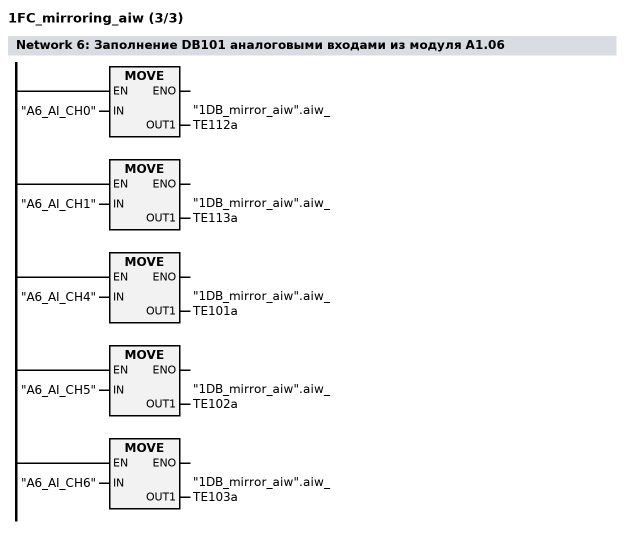
   RUNG wire#powerrail
      Move(in := "A6_AI_CH0", out1 => "1DB_mirror_aiw".aiw_TE112a)
   END_RUNG
   RUNG wire#powerrail
      Move(in := "A6_AI_CH1", out1 => "1DB_mirror_aiw".aiw_TE113a)
   END_RUNG
   RUNG wire#powerrail
      Move(in := "A6_AI_CH4", out1 => "1DB_mirror_aiw".aiw_TE101a)
   END_RUNG
   RUNG wire#powerrail
      Move(in := "A6_AI_CH5", out1 => "1DB_mirror_aiw".aiw_TE102a)
   END_RUNG
   RUNG wire#powerrail
      Move(in := "A6_AI_CH6", out1 => "1DB_mirror_aiw".aiw_TE103a)
   END_RUNG
   // the same network as SCL:
   "1DB_mirror_aiw".aiw_TE112a := "A6_AI_CH0";
   "1DB_mirror_aiw".aiw_TE113a := "A6_AI_CH1";
   "1DB_mirror_aiw".aiw_TE101a := "A6_AI_CH4";
   "1DB_mirror_aiw".aiw_TE102a := "A6_AI_CH5";
   "1DB_mirror_aiw".aiw_TE103a := "A6_AI_CH6";
END_REGION
END_FUNCTION

FUNCTION "1FC_mirroring_di" : Void   // FC102, LAD
{ S7_Optimized_Access := 'TRUE' }
VERSION : 0.1
// Эта функция безусловно заполняет блок данных 102 битами, соответствущими дискретным входам этого ПЛК. Другие прогаммы этого ПЛК читают исключительно DB102 и не читают непосредственно модули ввода дискретных сигналов
BEGIN

REGION Network 2: Заполнение DB102 дискретными входами из модуля А1.07
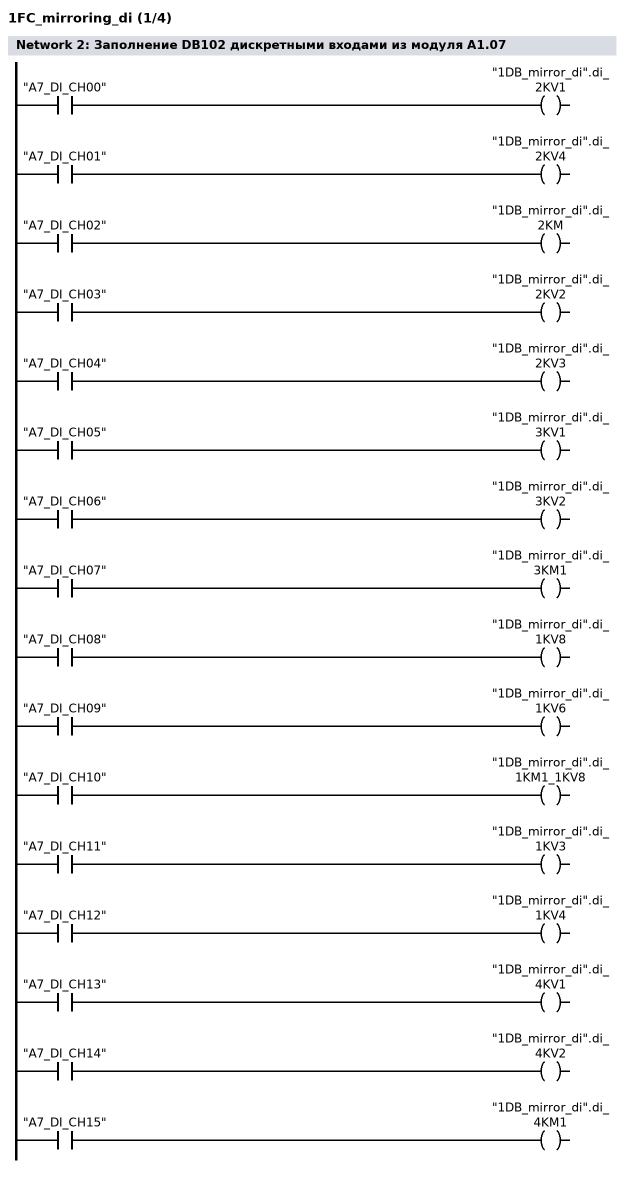
   RUNG wire#powerrail
      Contact( "A7_DI_CH00" )
      Coil( "1DB_mirror_di".di_2KV1 )
   END_RUNG
   RUNG wire#powerrail
      Contact( "A7_DI_CH01" )
      Coil( "1DB_mirror_di".di_2KV4 )
   END_RUNG
   RUNG wire#powerrail
      Contact( "A7_DI_CH02" )
      Coil( "1DB_mirror_di".di_2KM )
   END_RUNG
   RUNG wire#powerrail
      Contact( "A7_DI_CH03" )
      Coil( "1DB_mirror_di".di_2KV2 )
   END_RUNG
   RUNG wire#powerrail
      Contact( "A7_DI_CH04" )
      Coil( "1DB_mirror_di".di_2KV3 )
   END_RUNG
   RUNG wire#powerrail
      Contact( "A7_DI_CH05" )
      Coil( "1DB_mirror_di".di_3KV1 )
   END_RUNG
   RUNG wire#powerrail
      Contact( "A7_DI_CH06" )
      Coil( "1DB_mirror_di".di_3KV2 )
   END_RUNG
   RUNG wire#powerrail
      Contact( "A7_DI_CH07" )
      Coil( "1DB_mirror_di".di_3KM1 )
   END_RUNG
   RUNG wire#powerrail
      Contact( "A7_DI_CH08" )
      Coil( "1DB_mirror_di".di_1KV8 )
   END_RUNG
   RUNG wire#powerrail
      Contact( "A7_DI_CH09" )
      Coil( "1DB_mirror_di".di_1KV6 )
   END_RUNG
   RUNG wire#powerrail
      Contact( "A7_DI_CH10" )
      Coil( "1DB_mirror_di".di_1KM1_1KV8 )
   END_RUNG
   RUNG wire#powerrail
      Contact( "A7_DI_CH11" )
      Coil( "1DB_mirror_di".di_1KV3 )
   END_RUNG
   RUNG wire#powerrail
      Contact( "A7_DI_CH12" )
      Coil( "1DB_mirror_di".di_1KV4 )
   END_RUNG
   RUNG wire#powerrail
      Contact( "A7_DI_CH13" )
      Coil( "1DB_mirror_di".di_4KV1 )
   END_RUNG
   RUNG wire#powerrail
      Contact( "A7_DI_CH14" )
      Coil( "1DB_mirror_di".di_4KV2 )
   END_RUNG
   RUNG wire#powerrail
      Contact( "A7_DI_CH15" )
      Coil( "1DB_mirror_di".di_4KM1 )
   END_RUNG
   // the same network as SCL:
   "1DB_mirror_di".di_2KV1 := "A7_DI_CH00";
   "1DB_mirror_di".di_2KV4 := "A7_DI_CH01";
   "1DB_mirror_di".di_2KM := "A7_DI_CH02";
   "1DB_mirror_di".di_2KV2 := "A7_DI_CH03";
   "1DB_mirror_di".di_2KV3 := "A7_DI_CH04";
   "1DB_mirror_di".di_3KV1 := "A7_DI_CH05";
   "1DB_mirror_di".di_3KV2 := "A7_DI_CH06";
   "1DB_mirror_di".di_3KM1 := "A7_DI_CH07";
   "1DB_mirror_di".di_1KV8 := "A7_DI_CH08";
   "1DB_mirror_di".di_1KV6 := "A7_DI_CH09";
   "1DB_mirror_di".di_1KM1_1KV8 := "A7_DI_CH10";
   "1DB_mirror_di".di_1KV3 := "A7_DI_CH11";
   "1DB_mirror_di".di_1KV4 := "A7_DI_CH12";
   "1DB_mirror_di".di_4KV1 := "A7_DI_CH13";
   "1DB_mirror_di".di_4KV2 := "A7_DI_CH14";
   "1DB_mirror_di".di_4KM1 := "A7_DI_CH15";
END_REGION

REGION Network 3: Заполнение DB102 дискретными входами из модуля А1.08
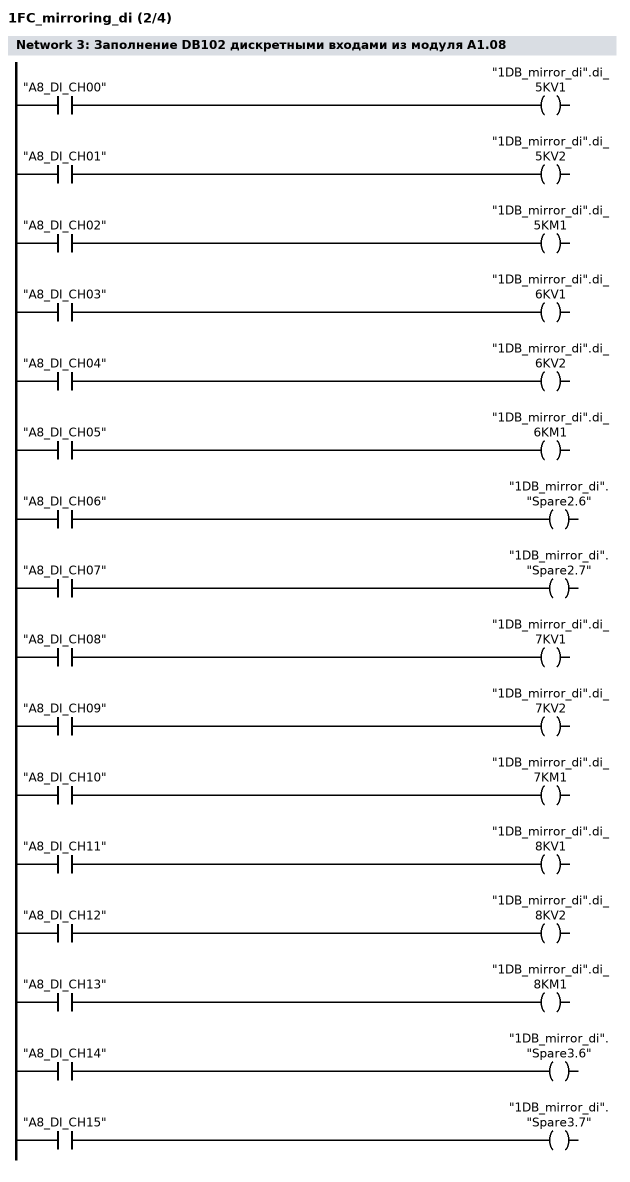
   RUNG wire#powerrail
      Contact( "A8_DI_CH00" )
      Coil( "1DB_mirror_di".di_5KV1 )
   END_RUNG
   RUNG wire#powerrail
      Contact( "A8_DI_CH01" )
      Coil( "1DB_mirror_di".di_5KV2 )
   END_RUNG
   RUNG wire#powerrail
      Contact( "A8_DI_CH02" )
      Coil( "1DB_mirror_di".di_5KM1 )
   END_RUNG
   RUNG wire#powerrail
      Contact( "A8_DI_CH03" )
      Coil( "1DB_mirror_di".di_6KV1 )
   END_RUNG
   RUNG wire#powerrail
      Contact( "A8_DI_CH04" )
      Coil( "1DB_mirror_di".di_6KV2 )
   END_RUNG
   RUNG wire#powerrail
      Contact( "A8_DI_CH05" )
      Coil( "1DB_mirror_di".di_6KM1 )
   END_RUNG
   RUNG wire#powerrail
      Contact( "A8_DI_CH06" )
      Coil( "1DB_mirror_di"."Spare2.6" )
   END_RUNG
   RUNG wire#powerrail
      Contact( "A8_DI_CH07" )
      Coil( "1DB_mirror_di"."Spare2.7" )
   END_RUNG
   RUNG wire#powerrail
      Contact( "A8_DI_CH08" )
      Coil( "1DB_mirror_di".di_7KV1 )
   END_RUNG
   RUNG wire#powerrail
      Contact( "A8_DI_CH09" )
      Coil( "1DB_mirror_di".di_7KV2 )
   END_RUNG
   RUNG wire#powerrail
      Contact( "A8_DI_CH10" )
      Coil( "1DB_mirror_di".di_7KM1 )
   END_RUNG
   RUNG wire#powerrail
      Contact( "A8_DI_CH11" )
      Coil( "1DB_mirror_di".di_8KV1 )
   END_RUNG
   RUNG wire#powerrail
      Contact( "A8_DI_CH12" )
      Coil( "1DB_mirror_di".di_8KV2 )
   END_RUNG
   RUNG wire#powerrail
      Contact( "A8_DI_CH13" )
      Coil( "1DB_mirror_di".di_8KM1 )
   END_RUNG
   RUNG wire#powerrail
      Contact( "A8_DI_CH14" )
      Coil( "1DB_mirror_di"."Spare3.6" )
   END_RUNG
   RUNG wire#powerrail
      Contact( "A8_DI_CH15" )
      Coil( "1DB_mirror_di"."Spare3.7" )
   END_RUNG
   // the same network as SCL:
   "1DB_mirror_di".di_5KV1 := "A8_DI_CH00";
   "1DB_mirror_di".di_5KV2 := "A8_DI_CH01";
   "1DB_mirror_di".di_5KM1 := "A8_DI_CH02";
   "1DB_mirror_di".di_6KV1 := "A8_DI_CH03";
   "1DB_mirror_di".di_6KV2 := "A8_DI_CH04";
   "1DB_mirror_di".di_6KM1 := "A8_DI_CH05";
   "1DB_mirror_di"."Spare2.6" := "A8_DI_CH06";
   "1DB_mirror_di"."Spare2.7" := "A8_DI_CH07";
   "1DB_mirror_di".di_7KV1 := "A8_DI_CH08";
   "1DB_mirror_di".di_7KV2 := "A8_DI_CH09";
   "1DB_mirror_di".di_7KM1 := "A8_DI_CH10";
   "1DB_mirror_di".di_8KV1 := "A8_DI_CH11";
   "1DB_mirror_di".di_8KV2 := "A8_DI_CH12";
   "1DB_mirror_di".di_8KM1 := "A8_DI_CH13";
   "1DB_mirror_di"."Spare3.6" := "A8_DI_CH14";
   "1DB_mirror_di"."Spare3.7" := "A8_DI_CH15";
END_REGION

REGION Network 4: Заполнение DB102 дискретными входами из модуля А1.09
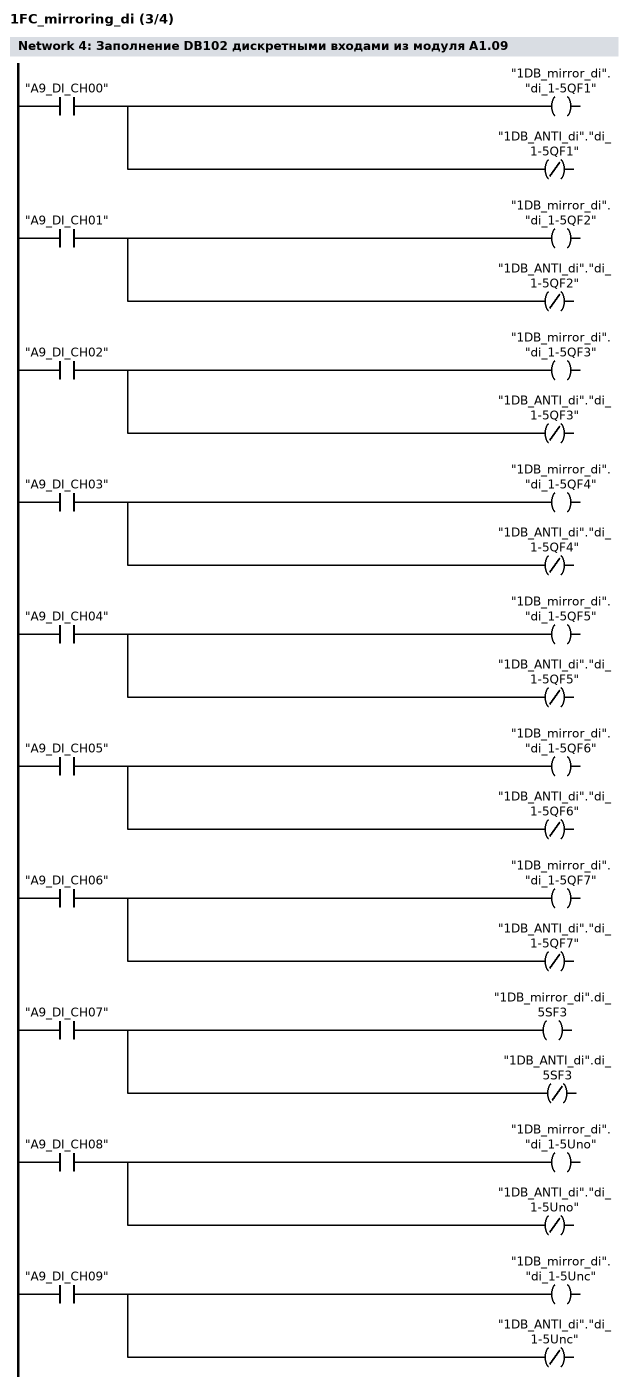
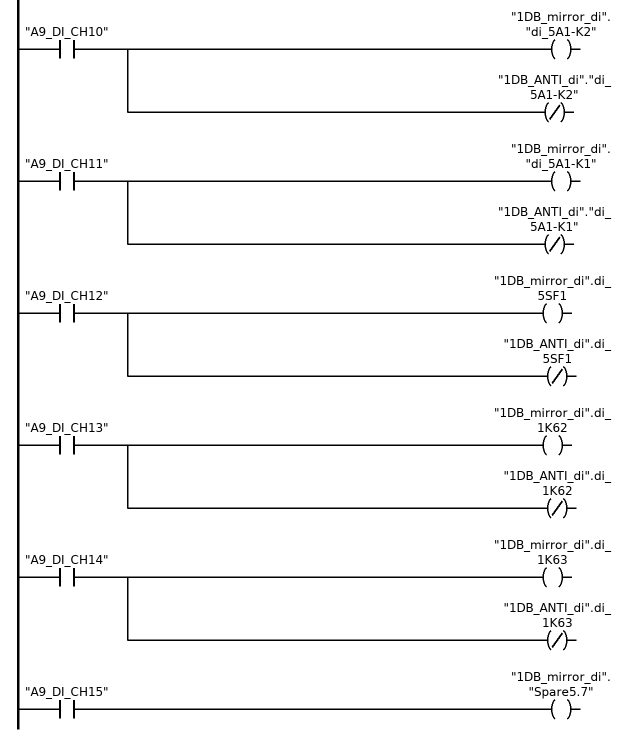
   RUNG wire#powerrail
      Contact( "A9_DI_CH00" )
      wire#w1
      Coil( "1DB_mirror_di"."di_1-5QF1" )
   END_RUNG
   RUNG wire#w1
      I_Coil( "1DB_ANTI_di"."di_1-5QF1" )
   END_RUNG
   RUNG wire#powerrail
      Contact( "A9_DI_CH01" )
      wire#w2
      Coil( "1DB_mirror_di"."di_1-5QF2" )
   END_RUNG
   RUNG wire#w2
      I_Coil( "1DB_ANTI_di"."di_1-5QF2" )
   END_RUNG
   RUNG wire#powerrail
      Contact( "A9_DI_CH02" )
      wire#w3
      Coil( "1DB_mirror_di"."di_1-5QF3" )
   END_RUNG
   RUNG wire#w3
      I_Coil( "1DB_ANTI_di"."di_1-5QF3" )
   END_RUNG
   RUNG wire#powerrail
      Contact( "A9_DI_CH03" )
      wire#w4
      Coil( "1DB_mirror_di"."di_1-5QF4" )
   END_RUNG
   RUNG wire#w4
      I_Coil( "1DB_ANTI_di"."di_1-5QF4" )
   END_RUNG
   RUNG wire#powerrail
      Contact( "A9_DI_CH04" )
      wire#w5
      Coil( "1DB_mirror_di"."di_1-5QF5" )
   END_RUNG
   RUNG wire#w5
      I_Coil( "1DB_ANTI_di"."di_1-5QF5" )
   END_RUNG
   RUNG wire#powerrail
      Contact( "A9_DI_CH05" )
      wire#w6
      Coil( "1DB_mirror_di"."di_1-5QF6" )
   END_RUNG
   RUNG wire#w6
      I_Coil( "1DB_ANTI_di"."di_1-5QF6" )
   END_RUNG
   RUNG wire#powerrail
      Contact( "A9_DI_CH06" )
      wire#w7
      Coil( "1DB_mirror_di"."di_1-5QF7" )
   END_RUNG
   RUNG wire#w7
      I_Coil( "1DB_ANTI_di"."di_1-5QF7" )
   END_RUNG
   RUNG wire#powerrail
      Contact( "A9_DI_CH07" )
      wire#w8
      Coil( "1DB_mirror_di".di_5SF3 )
   END_RUNG
   RUNG wire#w8
      I_Coil( "1DB_ANTI_di".di_5SF3 )
   END_RUNG
   RUNG wire#powerrail
      Contact( "A9_DI_CH08" )
      wire#w9
      Coil( "1DB_mirror_di"."di_1-5Uno" )
   END_RUNG
   RUNG wire#w9
      I_Coil( "1DB_ANTI_di"."di_1-5Uno" )
   END_RUNG
   RUNG wire#powerrail
      Contact( "A9_DI_CH09" )
      wire#w10
      Coil( "1DB_mirror_di"."di_1-5Unc" )
   END_RUNG
   RUNG wire#w10
      I_Coil( "1DB_ANTI_di"."di_1-5Unc" )
   END_RUNG
   RUNG wire#powerrail
      Contact( "A9_DI_CH10" )
      wire#w11
      Coil( "1DB_mirror_di"."di_5A1-K2" )
   END_RUNG
   RUNG wire#w11
      I_Coil( "1DB_ANTI_di"."di_5A1-K2" )
   END_RUNG
   RUNG wire#powerrail
      Contact( "A9_DI_CH11" )
      wire#w12
      Coil( "1DB_mirror_di"."di_5A1-K1" )
   END_RUNG
   RUNG wire#w12
      I_Coil( "1DB_ANTI_di"."di_5A1-K1" )
   END_RUNG
   RUNG wire#powerrail
      Contact( "A9_DI_CH12" )
      wire#w13
      Coil( "1DB_mirror_di".di_5SF1 )
   END_RUNG
   RUNG wire#w13
      I_Coil( "1DB_ANTI_di".di_5SF1 )
   END_RUNG
   RUNG wire#powerrail
      Contact( "A9_DI_CH13" )
      wire#w14
      Coil( "1DB_mirror_di".di_1K62 )
   END_RUNG
   RUNG wire#w14
      I_Coil( "1DB_ANTI_di".di_1K62 )
   END_RUNG
   RUNG wire#powerrail
      Contact( "A9_DI_CH14" )
      wire#w15
      Coil( "1DB_mirror_di".di_1K63 )
   END_RUNG
   RUNG wire#w15
      I_Coil( "1DB_ANTI_di".di_1K63 )
   END_RUNG
   RUNG wire#powerrail
      Contact( "A9_DI_CH15" )
      Coil( "1DB_mirror_di"."Spare5.7" )
   END_RUNG
   // the same network as SCL:
   "1DB_mirror_di"."di_1-5QF1" := "A9_DI_CH00";
   "1DB_ANTI_di"."di_1-5QF1" := NOT "A9_DI_CH00";
   "1DB_mirror_di"."di_1-5QF2" := "A9_DI_CH01";
   "1DB_ANTI_di"."di_1-5QF2" := NOT "A9_DI_CH01";
   "1DB_mirror_di"."di_1-5QF3" := "A9_DI_CH02";
   "1DB_ANTI_di"."di_1-5QF3" := NOT "A9_DI_CH02";
   "1DB_mirror_di"."di_1-5QF4" := "A9_DI_CH03";
   "1DB_ANTI_di"."di_1-5QF4" := NOT "A9_DI_CH03";
   "1DB_mirror_di"."di_1-5QF5" := "A9_DI_CH04";
   "1DB_ANTI_di"."di_1-5QF5" := NOT "A9_DI_CH04";
   "1DB_mirror_di"."di_1-5QF6" := "A9_DI_CH05";
   "1DB_ANTI_di"."di_1-5QF6" := NOT "A9_DI_CH05";
   "1DB_mirror_di"."di_1-5QF7" := "A9_DI_CH06";
   "1DB_ANTI_di"."di_1-5QF7" := NOT "A9_DI_CH06";
   "1DB_mirror_di".di_5SF3 := "A9_DI_CH07";
   "1DB_ANTI_di".di_5SF3 := NOT "A9_DI_CH07";
   "1DB_mirror_di"."di_1-5Uno" := "A9_DI_CH08";
   "1DB_ANTI_di"."di_1-5Uno" := NOT "A9_DI_CH08";
   "1DB_mirror_di"."di_1-5Unc" := "A9_DI_CH09";
   "1DB_ANTI_di"."di_1-5Unc" := NOT "A9_DI_CH09";
   "1DB_mirror_di"."di_5A1-K2" := "A9_DI_CH10";
   "1DB_ANTI_di"."di_5A1-K2" := NOT "A9_DI_CH10";
   "1DB_mirror_di"."di_5A1-K1" := "A9_DI_CH11";
   "1DB_ANTI_di"."di_5A1-K1" := NOT "A9_DI_CH11";
   "1DB_mirror_di".di_5SF1 := "A9_DI_CH12";
   "1DB_ANTI_di".di_5SF1 := NOT "A9_DI_CH12";
   "1DB_mirror_di".di_1K62 := "A9_DI_CH13";
   "1DB_ANTI_di".di_1K62 := NOT "A9_DI_CH13";
   "1DB_mirror_di".di_1K63 := "A9_DI_CH14";
   "1DB_ANTI_di".di_1K63 := NOT "A9_DI_CH14";
   "1DB_mirror_di"."Spare5.7" := "A9_DI_CH15";
END_REGION

REGION Network 6: Заполнение DB102 дискретными входами из CPU A1.01
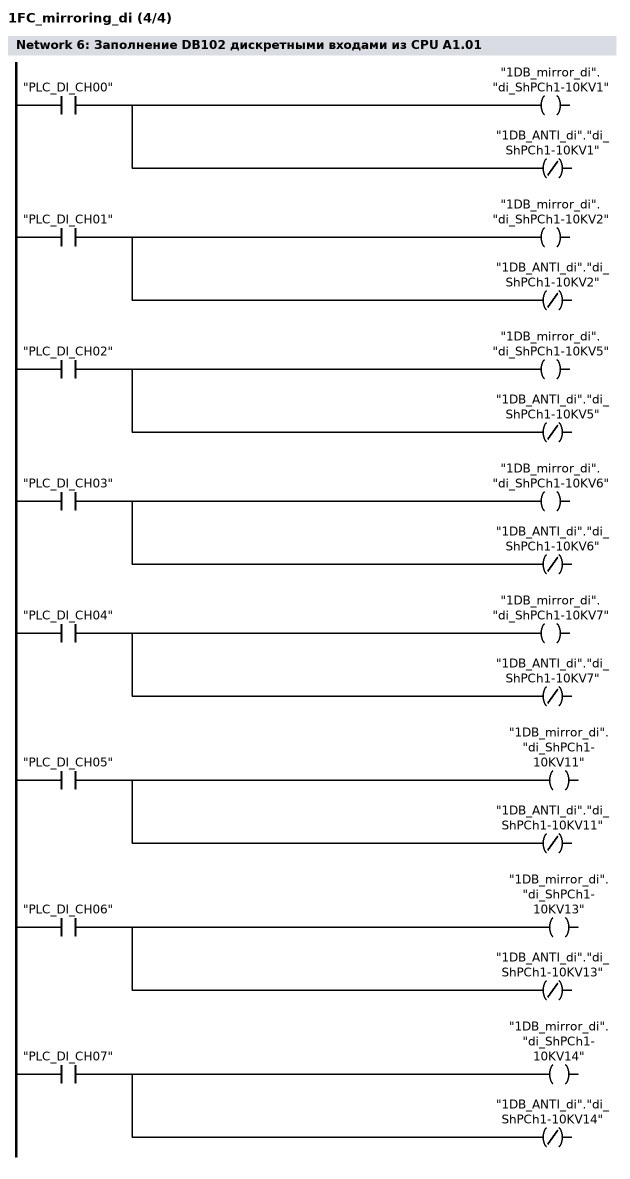
   RUNG wire#powerrail
      Contact( "PLC_DI_CH00" )
      wire#w1
      Coil( "1DB_mirror_di"."di_ShPCh1-10KV1" )
   END_RUNG
   RUNG wire#w1
      I_Coil( "1DB_ANTI_di"."di_ShPCh1-10KV1" )
   END_RUNG
   RUNG wire#powerrail
      Contact( "PLC_DI_CH01" )
      wire#w2
      Coil( "1DB_mirror_di"."di_ShPCh1-10KV2" )
   END_RUNG
   RUNG wire#w2
      I_Coil( "1DB_ANTI_di"."di_ShPCh1-10KV2" )
   END_RUNG
   RUNG wire#powerrail
      Contact( "PLC_DI_CH02" )
      wire#w3
      Coil( "1DB_mirror_di"."di_ShPCh1-10KV5" )
   END_RUNG
   RUNG wire#w3
      I_Coil( "1DB_ANTI_di"."di_ShPCh1-10KV5" )
   END_RUNG
   RUNG wire#powerrail
      Contact( "PLC_DI_CH03" )
      wire#w4
      Coil( "1DB_mirror_di"."di_ShPCh1-10KV6" )
   END_RUNG
   RUNG wire#w4
      I_Coil( "1DB_ANTI_di"."di_ShPCh1-10KV6" )
   END_RUNG
   RUNG wire#powerrail
      Contact( "PLC_DI_CH04" )
      wire#w5
      Coil( "1DB_mirror_di"."di_ShPCh1-10KV7" )
   END_RUNG
   RUNG wire#w5
      I_Coil( "1DB_ANTI_di"."di_ShPCh1-10KV7" )
   END_RUNG
   RUNG wire#powerrail
      Contact( "PLC_DI_CH05" )
      wire#w6
      Coil( "1DB_mirror_di"."di_ShPCh1-10KV11" )
   END_RUNG
   RUNG wire#w6
      I_Coil( "1DB_ANTI_di"."di_ShPCh1-10KV11" )
   END_RUNG
   RUNG wire#powerrail
      Contact( "PLC_DI_CH06" )
      wire#w7
      Coil( "1DB_mirror_di"."di_ShPCh1-10KV13" )
   END_RUNG
   RUNG wire#w7
      I_Coil( "1DB_ANTI_di"."di_ShPCh1-10KV13" )
   END_RUNG
   RUNG wire#powerrail
      Contact( "PLC_DI_CH07" )
      wire#w8
      Coil( "1DB_mirror_di"."di_ShPCh1-10KV14" )
   END_RUNG
   RUNG wire#w8
      I_Coil( "1DB_ANTI_di"."di_ShPCh1-10KV14" )
   END_RUNG
   // the same network as SCL:
   "1DB_mirror_di"."di_ShPCh1-10KV1" := "PLC_DI_CH00";
   "1DB_ANTI_di"."di_ShPCh1-10KV1" := NOT "PLC_DI_CH00";
   "1DB_mirror_di"."di_ShPCh1-10KV2" := "PLC_DI_CH01";
   "1DB_ANTI_di"."di_ShPCh1-10KV2" := NOT "PLC_DI_CH01";
   "1DB_mirror_di"."di_ShPCh1-10KV5" := "PLC_DI_CH02";
   "1DB_ANTI_di"."di_ShPCh1-10KV5" := NOT "PLC_DI_CH02";
   "1DB_mirror_di"."di_ShPCh1-10KV6" := "PLC_DI_CH03";
   "1DB_ANTI_di"."di_ShPCh1-10KV6" := NOT "PLC_DI_CH03";
   "1DB_mirror_di"."di_ShPCh1-10KV7" := "PLC_DI_CH04";
   "1DB_ANTI_di"."di_ShPCh1-10KV7" := NOT "PLC_DI_CH04";
   "1DB_mirror_di"."di_ShPCh1-10KV11" := "PLC_DI_CH05";
   "1DB_ANTI_di"."di_ShPCh1-10KV11" := NOT "PLC_DI_CH05";
   "1DB_mirror_di"."di_ShPCh1-10KV13" := "PLC_DI_CH06";
   "1DB_ANTI_di"."di_ShPCh1-10KV13" := NOT "PLC_DI_CH06";
   "1DB_mirror_di"."di_ShPCh1-10KV14" := "PLC_DI_CH07";
   "1DB_ANTI_di"."di_ShPCh1-10KV14" := NOT "PLC_DI_CH07";
END_REGION
END_FUNCTION

FUNCTION "1FC_mirroring_do" : Void   // FC103, LAD
{ S7_Optimized_Access := 'TRUE' }
VERSION : 0.1
// Эта функция безусловно пишет в дискретные выходы этого ПЛК биты, соответствущие битами из блока данных 103. Другие прогаммы этого ПЛК пишут исключительно в DB103 и не пишут непосредственно в модули вывода дискретных сигналов
BEGIN

REGION Network 2: Выгрузка дискретных выходов из DB103 в модуль A1.07
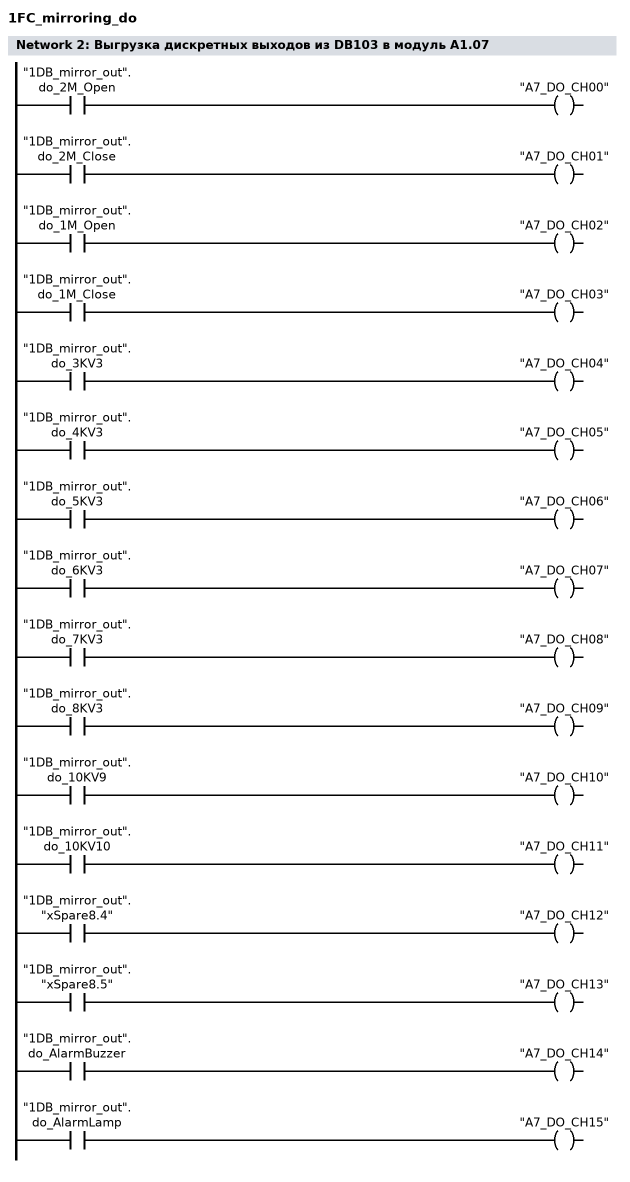
   RUNG wire#powerrail
      Contact( "1DB_mirror_out".do_2M_Open )
      Coil( "A7_DO_CH00" )
   END_RUNG
   RUNG wire#powerrail
      Contact( "1DB_mirror_out".do_2M_Close )
      Coil( "A7_DO_CH01" )
   END_RUNG
   RUNG wire#powerrail
      Contact( "1DB_mirror_out".do_1M_Open )
      Coil( "A7_DO_CH02" )
   END_RUNG
   RUNG wire#powerrail
      Contact( "1DB_mirror_out".do_1M_Close )
      Coil( "A7_DO_CH03" )
   END_RUNG
   RUNG wire#powerrail
      Contact( "1DB_mirror_out".do_3KV3 )
      Coil( "A7_DO_CH04" )
   END_RUNG
   RUNG wire#powerrail
      Contact( "1DB_mirror_out".do_4KV3 )
      Coil( "A7_DO_CH05" )
   END_RUNG
   RUNG wire#powerrail
      Contact( "1DB_mirror_out".do_5KV3 )
      Coil( "A7_DO_CH06" )
   END_RUNG
   RUNG wire#powerrail
      Contact( "1DB_mirror_out".do_6KV3 )
      Coil( "A7_DO_CH07" )
   END_RUNG
   RUNG wire#powerrail
      Contact( "1DB_mirror_out".do_7KV3 )
      Coil( "A7_DO_CH08" )
   END_RUNG
   RUNG wire#powerrail
      Contact( "1DB_mirror_out".do_8KV3 )
      Coil( "A7_DO_CH09" )
   END_RUNG
   RUNG wire#powerrail
      Contact( "1DB_mirror_out".do_10KV9 )
      Coil( "A7_DO_CH10" )
   END_RUNG
   RUNG wire#powerrail
      Contact( "1DB_mirror_out".do_10KV10 )
      Coil( "A7_DO_CH11" )
   END_RUNG
   RUNG wire#powerrail
      Contact( "1DB_mirror_out"."xSpare8.4" )
      Coil( "A7_DO_CH12" )
   END_RUNG
   RUNG wire#powerrail
      Contact( "1DB_mirror_out"."xSpare8.5" )
      Coil( "A7_DO_CH13" )
   END_RUNG
   RUNG wire#powerrail
      Contact( "1DB_mirror_out".do_AlarmBuzzer )
      Coil( "A7_DO_CH14" )
   END_RUNG
   RUNG wire#powerrail
      Contact( "1DB_mirror_out".do_AlarmLamp )
      Coil( "A7_DO_CH15" )
   END_RUNG
   // the same network as SCL:
   "A7_DO_CH00" := "1DB_mirror_out".do_2M_Open;
   "A7_DO_CH01" := "1DB_mirror_out".do_2M_Close;
   "A7_DO_CH02" := "1DB_mirror_out".do_1M_Open;
   "A7_DO_CH03" := "1DB_mirror_out".do_1M_Close;
   "A7_DO_CH04" := "1DB_mirror_out".do_3KV3;
   "A7_DO_CH05" := "1DB_mirror_out".do_4KV3;
   "A7_DO_CH06" := "1DB_mirror_out".do_5KV3;
   "A7_DO_CH07" := "1DB_mirror_out".do_6KV3;
   "A7_DO_CH08" := "1DB_mirror_out".do_7KV3;
   "A7_DO_CH09" := "1DB_mirror_out".do_8KV3;
   "A7_DO_CH10" := "1DB_mirror_out".do_10KV9;
   "A7_DO_CH11" := "1DB_mirror_out".do_10KV10;
   "A7_DO_CH12" := "1DB_mirror_out"."xSpare8.4";
   "A7_DO_CH13" := "1DB_mirror_out"."xSpare8.5";
   "A7_DO_CH14" := "1DB_mirror_out".do_AlarmBuzzer;
   "A7_DO_CH15" := "1DB_mirror_out".do_AlarmLamp;
END_REGION

REGION Network 3: Выгрузка дискретных выходов из DB103 в модуль A1.08
END_REGION

REGION Network 4: Выгрузка дискретных выходов из DB103 в модуль A1.09
END_REGION

REGION Network 5: Выгрузка дискретных выходов из DB103 в CPU A1.01
END_REGION
END_FUNCTION

FUNCTION "1FC_mirroring_aqw" : Void   // FC109, LAD
{ S7_Optimized_Access := 'TRUE' }
VERSION : 0.1
BEGIN

REGION Network 2: Выгрузка аналоговых выходов из DB103 в CPU A1.01
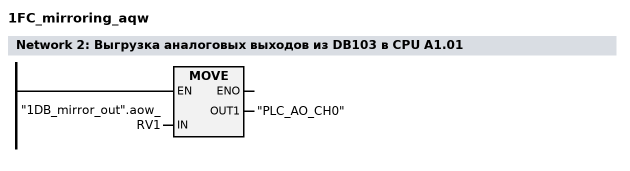
   RUNG wire#powerrail
      Move(in := "1DB_mirror_out".aow_RV1, out1 => "PLC_AO_CH0")
   END_RUNG
   // the same network as SCL:
   "PLC_AO_CH0" := "1DB_mirror_out".aow_RV1;
END_REGION
END_FUNCTION

// folder: Processing_AIO

FUNCTION_BLOCK "1FC_Compare"   // FB101, LAD
TITLE = Аварийные и предупредительные границы
{ S7_Optimized_Access := 'TRUE' }
VERSION : 0.1
// Функ.блок аварийных и предупредительных границ
   VAR_INPUT
      irTag : Real;   // Контролируемый параметр
      iiTag : Int;   // Контролируемый параметр, код АЦП
   END_VAR
   VAR_OUTPUT
      oxHWarning : Bool;   // Достигнута ВПГ
      oxLWarning : Bool;   // Достигнута НПГ
      oxHAlarm : Bool;   // Достигнута ВАГ
      oxLAlarm : Bool;   // Достигнута НАГ
      oxError : Bool;   // Вне диапазона модуля
   END_VAR
   VAR_IN_OUT
      iouWarning : "uWrnngAlarm";
      iouAlarm : "uWrnngAlarm";
   END_VAR
   VAR
      IEC_Timer_LWarning : TON_TIME;
      IEC_Timer_HWarning : TON_TIME;
      IEC_Timer_LAlarm : TON_TIME;
      IEC_Timer_HAlarm : TON_TIME;
   END_VAR
   VAR_TEMP
      tiUp : Int;
      tiDown : Int;
   END_VAR
   VAR CONSTANT
      ciOverUp : Int := 1000;
      ciOverDown : Int := 1000;
      ciUp : Int := 32512;   // Максимум диапазона для ошибки канала аналогоаого входа
      ciDown : Int := -4865;   // Минимум диапазона для ошибки канала аналогоаого входа
   END_VAR
BEGIN

REGION Network 2 (SCL): Расчет пределов ошибки инженерного значения ан.входа в зависимости от бита
   IF "xSelectErrRange" THEN
       #tiDown := 0 - "iDeltaErrRangeDown"; //#ciOverDown;
       #tiUp := 27648 + "iDeltaErrRangeUp"; //#ciOverUp;
   ELSE
       #tiDown := #ciDown;
       #tiUp := #ciUp;
   END_IF;
   "iValueErrRangeMin" := #tiDown;
   "iValueErrRangeMax" := #tiUp;
END_REGION

REGION Network 3: Вне диапазона модуля
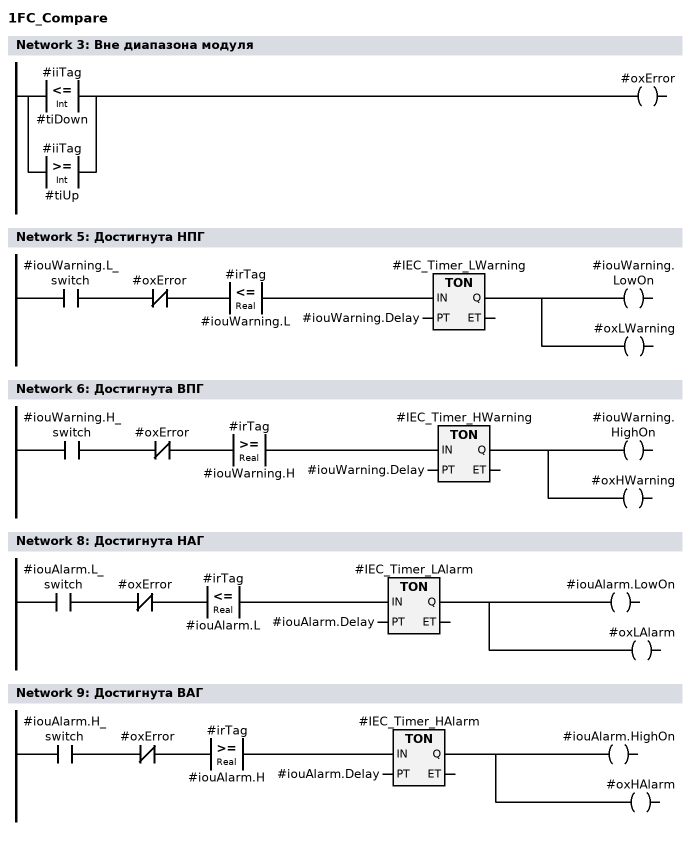
   RUNG wire#powerrail
      { S7_Templates := "SrcType := Int" } LE_Contact(in1 := #iiTag, in2 := #tiDown)
      wire#w1
      Coil( #oxError )
   END_RUNG
   RUNG wire#powerrail
      { S7_Templates := "SrcType := Int" } GE_Contact(in1 := #iiTag, in2 := #tiUp)
   END_RUNG wire#w1
   // the same network as SCL:
   #oxError := (#iiTag <= #tiDown) OR (#iiTag >= #tiUp);
END_REGION

REGION Network 5: Достигнута НПГ
   #IEC_Timer_LWarning(IN := #iouWarning.L_switch AND NOT #oxError AND (#irTag <= #iouWarning.L),   // TON
                       PT := #iouWarning.Delay);
   #iouWarning.LowOn := #IEC_Timer_LWarning.Q;
   #oxLWarning := #IEC_Timer_LWarning.Q;
END_REGION

REGION Network 6: Достигнута ВПГ
   #IEC_Timer_HWarning(IN := #iouWarning.H_switch AND NOT #oxError AND (#irTag >= #iouWarning.H),   // TON
                       PT := #iouWarning.Delay);
   #iouWarning.HighOn := #IEC_Timer_HWarning.Q;
   #oxHWarning := #IEC_Timer_HWarning.Q;
END_REGION

REGION Network 8: Достигнута НАГ
   #IEC_Timer_LAlarm(IN := #iouAlarm.L_switch AND NOT #oxError AND (#irTag <= #iouAlarm.L),   // TON
                     PT := #iouAlarm.Delay);
   #iouAlarm.LowOn := #IEC_Timer_LAlarm.Q;
   #oxLAlarm := #IEC_Timer_LAlarm.Q;
END_REGION

REGION Network 9: Достигнута ВАГ
   #IEC_Timer_HAlarm(IN := #iouAlarm.H_switch AND NOT #oxError AND (#irTag >= #iouAlarm.H),   // TON
                     PT := #iouAlarm.Delay);
   #iouAlarm.HighOn := #IEC_Timer_HAlarm.Q;
   #oxHAlarm := #IEC_Timer_HAlarm.Q;
END_REGION
END_FUNCTION_BLOCK

FUNCTION_BLOCK "1FB_Control"   // FB113, LAD
TITLE = Проверка аналогового входа на авар.и предупр.границы
{ S7_Optimized_Access := 'TRUE' }
VERSION : 0.1
// Функ.блок проверки аналогового входа на предупр.и аварийные границы
   VAR_INPUT
      irTag : Real;   // Контролируемый параметр
      iiTag : Int;   // Контролируемый параметр, код АЦП
   END_VAR
   VAR_OUTPUT
      owCode : Word;   // Равно 0, если все хорошо
      oxFault : Bool;   // Авария датчика
   END_VAR
   VAR_IN_OUT
      iouWarning : "uWrnngAlarm";   // Структура предупреждений
      iouAlarm : "uWrnngAlarm";   // Структура аварий
   END_VAR
   VAR
      suCompare_Instance : "1FC_Compare";   // Экземпляр для FB101
   END_VAR
   VAR_TEMP
      txHWarning : Bool;   // Если ВПГ нарушена
      txLWarning : Bool;   // Если НПГ нарушена
      txHAlarm : Bool;   // Если ВАГ нарушена
      txLAlarm : Bool;   // Если НАГ нарушена
      txError : Bool;   // Если вне диапазона модуля
   END_VAR
   VAR_TEMP   // added for the SCL form of the ladder/FBD networks
      _w1 : Bool;
   END_VAR
BEGIN

REGION Network 2: Расчет (заполнение битами) слова состояния аналогового входа
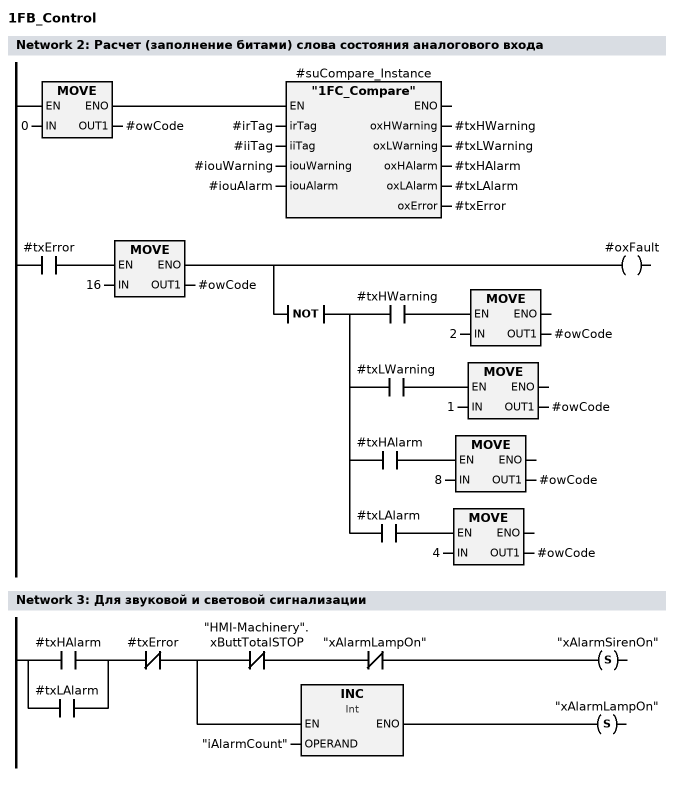
   RUNG wire#powerrail
      Move(in := 0, out1 => #owCode)
      #suCompare_Instance(irTag := #irTag, iiTag := #iiTag, iouWarning := #iouWarning, iouAlarm := #iouAlarm, oxHWarning => #txHWarning, oxLWarning => #txLWarning, oxHAlarm => #txHAlarm, oxLAlarm => #txLAlarm, oxError => #txError)
   END_RUNG
   RUNG wire#powerrail
      Contact( #txError )
      Move(in := 16, out1 => #owCode)
      wire#w1
      Coil( #oxFault )
   END_RUNG
   RUNG wire#w1
      Not()
      wire#w2
      Contact( #txHWarning )
      Move(in := 2, out1 => #owCode)
   END_RUNG
   RUNG wire#w2
      Contact( #txLWarning )
      Move(in := 1, out1 => #owCode)
   END_RUNG
   RUNG wire#w2
      Contact( #txHAlarm )
      Move(in := 8, out1 => #owCode)
   END_RUNG
   RUNG wire#w2
      Contact( #txLAlarm )
      Move(in := 4, out1 => #owCode)
   END_RUNG
   // the same network as SCL:
   #owCode := 0;
   #suCompare_Instance(irTag := #irTag,   // "1FC_Compare"
                       iiTag := #iiTag,
                       iouWarning := #iouWarning,
                       iouAlarm := #iouAlarm,
                       oxHWarning => #txHWarning,
                       oxLWarning => #txLWarning,
                       oxHAlarm => #txHAlarm,
                       oxLAlarm => #txLAlarm,
                       oxError => #txError);
   IF #txError THEN #owCode := 16; END_IF;
   #oxFault := #txError;
   IF NOT #txError AND #txHWarning THEN #owCode := 2; END_IF;
   IF NOT #txError AND #txLWarning THEN #owCode := 1; END_IF;
   IF NOT #txError AND #txHAlarm THEN #owCode := 8; END_IF;
   IF NOT #txError AND #txLAlarm THEN #owCode := 4; END_IF;
END_REGION

REGION Network 3: Для звуковой и световой сигнализации
   RUNG wire#powerrail
      Contact( #txHAlarm )
      wire#w1
      I_Contact( #txError )
      wire#w2
      I_Contact( "HMI-Machinery".xButtTotalSTOP )
      I_Contact( "xAlarmLampOn" )
      S_Coil( "xAlarmSirenOn" )
   END_RUNG
   RUNG wire#powerrail
      Contact( #txLAlarm )
   END_RUNG wire#w1
   RUNG wire#w2
      { S7_Templates := "DestType := Int" } Inc( "iAlarmCount" )
      S_Coil( "xAlarmLampOn" )
   END_RUNG
   // the same network as SCL:
   #_w1 := (#txHAlarm OR #txLAlarm) AND NOT #txError;
   IF #_w1 AND NOT "HMI-Machinery".xButtTotalSTOP AND NOT "xAlarmLampOn" THEN
       "xAlarmSirenOn" := TRUE;
   END_IF;
   IF #_w1 THEN
       "iAlarmCount" := "iAlarmCount" + 1;
       "xAlarmLampOn" := TRUE;
   END_IF;
END_REGION
END_FUNCTION_BLOCK

FUNCTION_BLOCK "1FB_Scale"   // FB130, LAD
TITLE = Физ.значение аналогового входа
{ S7_Optimized_Access := 'TRUE' }
VERSION : 0.1
// Преорбазование аналогового входа в физ.значение согласно шкалы
   VAR_INPUT
      iiRaw : Int;   // Входной сигнал
      iuScale : "uScale";
   END_VAR
   VAR_OUTPUT
      orScaled : Real;   // Выходное отмасштабированное значение
   END_VAR
   VAR
      srLowPassLastFv : Real;   // Выходное значение для следующего цикла расчета
   END_VAR
   VAR_TEMP
      trValNormToScale : Real;   // Временная переменная
      txFilterZRError : Bool;   // Ошибка, если t = 0,0s
   END_VAR
BEGIN

REGION Network 2: Нормализация + масштабирование
